    // Sequence is advanced only when the actual command image changes.
    // This keeps the command stable long enough for adapter ACK validation.
    L_Command_Changed :=
        (L_Command_Enable <> L_Last_Command_Enable[L_i]) OR
        (L_Setpoint_x10 <> L_Last_Command_Setpoint_x10[L_i]);

    IF L_Command_Changed THEN
        GVL_OPENTHERM_ADAPTER.G_Command[L_i].Sequence :=
            GVL_OPENTHERM_ADAPTER.G_Command[L_i].Sequence + 1;

        GVL_OPENTHERM_ADAPTER.G_Command[L_i].Last_Write_MS :=
            GVL_STATUS.G_System_Time_MS;

        L_Last_Command_Enable[L_i] := L_Command_Enable;
        L_Last_Command_Setpoint_x10[L_i] := L_Setpoint_x10;
    END_IF;

    // Command is valid only when the adapter confirms the current stable sequence.
    VO_OT_Command_Valid[L_i] :=
        L_Command_Enable AND
        GVL_OPENTHERM_ADAPTER.G_Status[L_i].Command_Ack AND
        (NOT GVL_OPENTHERM_ADAPTER.G_Status[L_i].Adapter_Error) AND
        GVL_OPENTHERM_ADAPTER.G_Status[L_i].Adapter_Online;

END_FOR;
          
END_FUNCTION_BLOCK

FUNCTION_BLOCK FB_Heating_Source_Stability_Observer
  VAR_INPUT
    VI_Enable : BOOL;
    VI_System_Time_MS : UDINT;
  END_VAR
  VAR
    L_i : INT;
    L_Last_Confidence : ARRAY[1..GVL_CONSTANTS.C_MAX_HEATING_CIRCUITS] OF REAL;
    L_Confidence_Delta : REAL;
    L_Confidence_Volatility : REAL;
    L_Source_Trust_Trend : REAL;
    L_Instability_Score : REAL;
  END_VAR

            // ==============================================================================
// Heating source stability observer
//
// Predictive observability-only layer.
//
// DOES NOT own runtime authority.
// DOES NOT own outputs.
// DOES NOT close valves.
// DOES NOT modify heating demand.
// DOES NOT override runtime decisions.
//
// Observes:
// - source switching frequency
// - fallback oscillation
// - degradation persistence
// - recovery trends
// - confidence volatility
//
// Publishes predictive instability semantics only.
//
// Reads only canonical runtime projection contracts.
// Does not depend on explainability publication topology.
// ==============================================================================



IF NOT VI_Enable THEN
    RETURN;
END_IF;

FOR L_i := 1 TO GVL_CONSTANTS.C_MAX_HEATING_CIRCUITS DO

    // ======================================================
    // VISIBILITY
    // ======================================================
    GVL_Heating_Source_Stability.G_State[L_i].Visible :=
        GVL_Heating_Runtime_Projection.G_Circuit_Projection[L_i].Visible;

    // ======================================================
    // EDGE COUNTING
    // ======================================================
    IF GVL_Heating_Runtime_Projection.G_Circuit_Projection[L_i].Source_Switched_Event THEN
        IF GVL_Heating_Source_Stability.G_State[L_i].Source_Switch_Count < 65535 THEN
            GVL_Heating_Source_Stability.G_State[L_i].Source_Switch_Count :=
                GVL_Heating_Source_Stability.G_State[L_i].Source_Switch_Count + 1;
        END_IF;

        GVL_Heating_Source_Stability.G_State[L_i].Last_Observation_MS :=
            VI_System_Time_MS;
    END_IF;

    IF GVL_Heating_Runtime_Projection.G_Circuit_Projection[L_i].Fallback_Activated_Event THEN
        IF GVL_Heating_Source_Stability.G_State[L_i].Fallback_Activation_Count < 65535 THEN
            GVL_Heating_Source_Stability.G_State[L_i].Fallback_Activation_Count :=
                GVL_Heating_Source_Stability.G_State[L_i].Fallback_Activation_Count + 1;
        END_IF;

        GVL_Heating_Source_Stability.G_State[L_i].Last_Observation_MS :=
            VI_System_Time_MS;
    END_IF;

    IF GVL_Heating_Runtime_Projection.G_Circuit_Projection[L_i].Fallback_Recovered_Event THEN
        IF GVL_Heating_Source_Stability.G_State[L_i].Fallback_Recovery_Count < 65535 THEN
            GVL_Heating_Source_Stability.G_State[L_i].Fallback_Recovery_Count :=
                GVL_Heating_Source_Stability.G_State[L_i].Fallback_Recovery_Count + 1;
        END_IF;

        GVL_Heating_Source_Stability.G_State[L_i].Last_Observation_MS :=
            VI_System_Time_MS;
    END_IF;

    IF GVL_Heating_Runtime_Projection.G_Circuit_Projection[L_i].Source_Loss_Event THEN
        IF GVL_Heating_Source_Stability.G_State[L_i].Source_Loss_Count < 65535 THEN
            GVL_Heating_Source_Stability.G_State[L_i].Source_Loss_Count :=
                GVL_Heating_Source_Stability.G_State[L_i].Source_Loss_Count + 1;
        END_IF;

        GVL_Heating_Source_Stability.G_State[L_i].Last_Observation_MS :=
            VI_System_Time_MS;
    END_IF;

    // ======================================================
    // CONFIDENCE VOLATILITY
    // ======================================================
    L_Confidence_Delta := ABS(
        GVL_Heating_Runtime_Projection.G_Circuit_Projection[L_i].Selected_Source_Confidence -
        L_Last_Confidence[L_i]
    );

    L_Confidence_Volatility :=
        GVL_Heating_Source_Stability.G_State[L_i].Confidence_Volatility * REAL#0.90 +
        L_Confidence_Delta * REAL#0.10;

    IF L_Confidence_Volatility < REAL#0.0 THEN
        L_Confidence_Volatility := REAL#0.0;
    ELSIF L_Confidence_Volatility > REAL#1.0 THEN
        L_Confidence_Volatility := REAL#1.0;
    END_IF;

    GVL_Heating_Source_Stability.G_State[L_i].Confidence_Volatility :=
        L_Confidence_Volatility;

    // ======================================================
    // SOURCE TRUST TREND
    // ======================================================
    L_Source_Trust_Trend :=
        GVL_Heating_Source_Stability.G_State[L_i].Source_Trust_Trend * REAL#0.95 +
        GVL_Heating_Runtime_Projection.G_Circuit_Projection[L_i].Selected_Source_Confidence * REAL#0.05;

    IF GVL_Heating_Runtime_Projection.G_Circuit_Projection[L_i].Source_Degraded THEN
        L_Source_Trust_Trend := L_Source_Trust_Trend * REAL#0.98;
    END_IF;

    IF L_Source_Trust_Trend < REAL#0.0 THEN
        L_Source_Trust_Trend := REAL#0.0;
    ELSIF L_Source_Trust_Trend > REAL#1.0 THEN
        L_Source_Trust_Trend := REAL#1.0;
    END_IF;

    GVL_Heating_Source_Stability.G_State[L_i].Source_Trust_Trend :=
        L_Source_Trust_Trend;

    // ======================================================
    // TREND OBSERVATION
    // ======================================================
    GVL_Heating_Source_Stability.G_State[L_i].Degraded_Trend_Visible :=
        GVL_Heating_Runtime_Projection.G_Circuit_Projection[L_i].Source_Degraded OR
        (GVL_Heating_Source_Stability.G_State[L_i].Fallback_Activation_Count >
         GVL_Heating_Source_Stability.G_State[L_i].Fallback_Recovery_Count);

    GVL_Heating_Source_Stability.G_State[L_i].Recovery_Trend_Visible :=
        (GVL_Heating_Source_Stability.G_State[L_i].Fallback_Recovery_Count > 0) AND
        (GVL_Heating_Source_Stability.G_State[L_i].Fallback_Recovery_Count >=
         GVL_Heating_Source_Stability.G_State[L_i].Fallback_Activation_Count);

    GVL_Heating_Source_Stability.G_State[L_i].Oscillation_Detected :=
        (GVL_Heating_Source_Stability.G_State[L_i].Source_Switch_Count >= 3) OR
        ((GVL_Heating_Source_Stability.G_State[L_i].Fallback_Activation_Count >= 2) AND
         (GVL_Heating_Source_Stability.G_State[L_i].Fallback_Recovery_Count >= 2));

    // ======================================================
    // INSTABILITY SCORE
    // ======================================================
    L_Instability_Score := REAL#0.0;

    IF GVL_Heating_Source_Stability.G_State[L_i].Oscillation_Detected THEN
        L_Instability_Score := L_Instability_Score + REAL#40.0;
    END_IF;

    IF GVL_Heating_Source_Stability.G_State[L_i].Degraded_Trend_Visible THEN
        L_Instability_Score := L_Instability_Score + REAL#30.0;
    END_IF;

    IF GVL_Heating_Source_Stability.G_State[L_i].Source_Loss_Count > 0 THEN
        L_Instability_Score := L_Instability_Score + REAL#30.0;
    END_IF;

    L_Instability_Score :=
        L_Instability_Score +
        (GVL_Heating_Source_Stability.G_State[L_i].Confidence_Volatility * REAL#20.0);

    IF L_Instability_Score > REAL#100.0 THEN
        L_Instability_Score := REAL#100.0;
    END_IF;

    GVL_Heating_Source_Stability.G_State[L_i].Instability_Score :=
        L_Instability_Score;

    GVL_Heating_Source_Stability.G_State[L_i].Instability_Attention :=
        L_Instability_Score >= REAL#60.0;

    // ======================================================
    // EXPLAINABILITY PUBLICATION
    // ======================================================
    IF GVL_Heating_Source_Stability.G_State[L_i].Source_Loss_Count > 0 THEN
        GVL_Heating_Source_Stability.G_State[L_i].Status_Code := 904;
        GVL_Heating_Source_Stability.G_State[L_i].Status_Text :=
            'Predictive source instability: source loss observed';

    ELSIF GVL_Heating_Source_Stability.G_State[L_i].Oscillation_Detected THEN
        GVL_Heating_Source_Stability.G_State[L_i].Status_Code := 903;
        GVL_Heating_Source_Stability.G_State[L_i].Status_Text :=
            'Predictive source instability: oscillation detected';

    ELSIF GVL_Heating_Source_Stability.G_State[L_i].Degraded_Trend_Visible THEN
        GVL_Heating_Source_Stability.G_State[L_i].Status_Code := 902;
        GVL_Heating_Source_Stability.G_State[L_i].Status_Text :=
            'Predictive source degradation trend observed';

    ELSE
        GVL_Heating_Source_Stability.G_State[L_i].Status_Code := 901;
        GVL_Heating_Source_Stability.G_State[L_i].Status_Text :=
            'Source stability nominal';
    END_IF;

    L_Last_Confidence[L_i] :=
        GVL_Heating_Runtime_Projection.G_Circuit_Projection[L_i].Selected_Source_Confidence;
END_FOR;

// >>> BULK_SYNC_ANCHOR: FB_Heating_Source_Stability_Observer <<<
          
END_FUNCTION_BLOCK

FUNCTION_BLOCK FB_Config_Simulation
  VAR_INPUT
    VI_Enable : BOOL;
    VI_Request : BOOL;
    VI_Confirm : BOOL;
  END_VAR
  VAR_OUTPUT
    VO_Executed : BOOL;
    VO_Result_OK : BOOL;
    VO_Error_Text : STRING(200);
  END_VAR
  VAR
    L_Error : BOOL;
  END_VAR

            // ==============================================================================
// Config simulation / validation function block
// Service/commissioning validation utility.
// Does NOT own runtime control and does NOT participate in heating phase runtime.
// ==============================================================================



VO_Executed := FALSE;
VO_Result_OK := GVL_CONFIG_SIMULATION.G_Simulation_Result_OK;
VO_Error_Text := GVL_CONFIG_SIMULATION.G_Simulation_Error_Text;

IF NOT VI_Enable THEN
    RETURN;
END_IF;

IF VI_Request AND VI_Confirm THEN

    L_Error := FALSE;
    VO_Result_OK := TRUE;
    VO_Error_Text := '';

    // Simulate INPUT constraints
    IF (GVL_CONFIG_CONTROL.STG_Reputation_Learning_Rate < 0.0) OR (GVL_CONFIG_CONTROL.STG_Reputation_Learning_Rate > 1.0) THEN
        VO_Result_OK := FALSE;
        VO_Error_Text := 'Invalid learning rate';
        L_Error := TRUE;
    END_IF;

    // Simulate SCENARIO logic
    IF GVL_CONFIG_CONTROL.STG_Night_Start_Hour = GVL_CONFIG_CONTROL.STG_Night_End_Hour THEN
        VO_Result_OK := FALSE;
        VO_Error_Text := 'Night window invalid';
        L_Error := TRUE;
    END_IF;

    // Simulate SAFETY
    IF GVL_CONFIG_CONTROL.STG_Stabilization_Delay_MS < 1000 THEN
        VO_Result_OK := FALSE;
        VO_Error_Text := 'Recovery delay too small';
        L_Error := TRUE;
    END_IF;

    // Simulate FAIL-SAFE policy
    IF NOT (
        GVL_CONFIG_CONTROL.STG_PLC_Inactive_Close_Gas OR
        GVL_CONFIG_CONTROL.STG_PLC_Inactive_Stop_Boiler OR
        GVL_CONFIG_CONTROL.STG_PLC_Inactive_Block_Heating OR
        GVL_CONFIG_CONTROL.STG_PLC_Inactive_Stop_Vent OR
        GVL_CONFIG_CONTROL.STG_PLC_Inactive_Block_Water
    ) THEN
        VO_Result_OK := FALSE;
        VO_Error_Text := 'Fail-safe disabled';
        L_Error := TRUE;
    END_IF;

    GVL_CONFIG_SIMULATION.G_Simulation_Result_OK := NOT L_Error;
    GVL_CONFIG_SIMULATION.G_Simulation_Error_Text := VO_Error_Text;
    GVL_CONFIG_SIMULATION.G_Simulation_Last_Run_MS := GVL_TIME_SERVICE.G_Now_MS;
    VO_Executed := TRUE;

END_IF;

// >>> BULK_SYNC_ANCHOR: FB_Config_Simulation <<<
          
END_FUNCTION_BLOCK

FUNCTION_BLOCK FB_DHW_Manager
  VAR_INPUT
    VI_System_Time_MS : UDINT;
    VI_Current_TOD : TOD;
    VI_IsActivePLC : BOOL;
    VI_Temp : REAL;
    VI_Pressure : REAL;
    VI_Config : ST_DHW_Config;
    VI_Current_Day_Of_Week : UINT;
    VI_Reset_Errors : BOOL;
    VI_Emergency_Stop : BOOL;
    VI_System_Mode : E_System_Operating_Mode;
    VI_IO_Modules_Online : ARRAY[1..GVL_CONSTANTS.C_MAX_MODULES] OF BOOL;
  END_VAR
  VAR_OUTPUT
    VO_Status : ST_DHW_Status;
    VO_Heating_Pump : BOOL;
    VO_Circ_Pump : BOOL;
  END_VAR
  VAR
    L_i : INT;
    L_Current_TOD : TOD;
    L_Legionella_Active : BOOL;
    L_Legionella_Timer : FB_System_Timer;
    L_Last_Good_Temp : REAL := 55.0;
    L_Legionella_Done_Today : BOOL;
    L_Last_Legionella_Day : UINT;
    fbTempValidator : FB_Analog_Validator;
    fbPressValidator : FB_Analog_Validator;
    L_Error_Latched : BOOL;
    L_Error_ID_Latched : WORD;
    L_Policy_Degraded : BOOL;
    L_Policy_Freeze_Protection : BOOL;
    L_Policy_Safe_Stop : BOOL;
    L_Target_Temp_Adjusted : REAL;
  END_VAR

            // >>> SYNC_TEST_MARKER_001 <<<


IF NOT VI_IsActivePLC THEN RETURN; END_IF;


GVL_STATE.G_DHW_IO_Fault := FALSE;
GVL_STATE.G_DHW_Sensor_Fault := FALSE;
GVL_STATE.G_DHW_Subsystem_Degraded := FALSE;

IF VI_Emergency_Stop THEN
    VO_Heating_Pump := FALSE;
    VO_Circ_Pump := FALSE;
    VO_Status.Warning := FALSE;
    VO_Status.Error := TRUE;
    VO_Status.Error_ID := TO_WORD(GVL_CONFIG.ERR_DHW_IO_OFFLINE); // временно используем общий аварийный код до детализации safety-кодов
    VO_Status.Heating_Pump_On := FALSE;
    VO_Status.Circ_Pump_On := FALSE;
    RETURN;
END_IF;

// Фиксация текущего времени
L_Current_TOD := VI_Current_TOD;

// ========================================
// DHW POLICY LAYER
// ========================================
L_Policy_Safe_Stop := (VI_System_Mode = E_System_Operating_Mode.MODE_SAFE_STOP);
L_Policy_Freeze_Protection := (VI_System_Mode = E_System_Operating_Mode.MODE_FREEZE_PROTECTION);
L_Policy_Degraded := (VI_System_Mode = E_System_Operating_Mode.MODE_DEGRADED);
L_Target_Temp_Adjusted := VI_Config.Target_Temp;
IF L_Policy_Degraded THEN
    L_Target_Temp_Adjusted := VI_Config.Target_Temp - VI_Config.Degraded_Target_Delta;
END_IF;

// ========================================
// DHW POLICY OVERRIDE
// ========================================
IF L_Policy_Safe_Stop THEN
    VO_Heating_Pump := FALSE;
    VO_Circ_Pump := FALSE;
    RETURN;
END_IF;

IF L_Policy_Freeze_Protection THEN
    VO_Heating_Pump := FALSE;
    VO_Circ_Pump := FALSE;
    RETURN;
END_IF;

// Сброс признака выполнения термодезинфекции при смене дня.
IF L_Last_Legionella_Day <> VI_Current_Day_Of_Week THEN
    L_Legionella_Done_Today := FALSE;
    L_Last_Legionella_Day := VI_Current_Day_Of_Week;
END_IF;

// Базовый сброс незащёлкнутых статусных флагов на текущий цикл.
// Критические ошибки ниже могут зафиксироваться и завершить выполнение через RETURN.
VO_Status.Warning := FALSE;
VO_Status.Error := FALSE;
VO_Status.Error_ID := 0;

// Сброс ошибок
IF VI_Reset_Errors THEN
    L_Error_Latched := FALSE;
    L_Error_ID_Latched := 0;
END_IF;

// Проверка связи с модулями ввода-вывода
FOR L_i := 1 TO GVL_CONSTANTS.C_MAX_MODULES DO
    IF NOT VI_IO_Modules_Online[L_i] THEN
        L_Error_Latched := TRUE;
        GVL_STATE.G_DHW_IO_Fault := TRUE;
        L_Error_ID_Latched := TO_WORD(GVL_CONFIG.ERR_DHW_IO_OFFLINE); // Потеря связи с модулями ввода-вывода
    END_IF;
END_FOR;

// 1. Обработка неисправностей датчиков и сервисных режимов (ТЗ 7.0)
fbTempValidator(
    VI_Value := VI_Temp,
    VI_Min_Valid := 0.0,
    VI_Max_Valid := 100.0,
    VI_Fallback_Mode := 0,
    VI_Default_Value := 55.0
);

fbPressValidator(
    VI_Value := VI_Pressure,
    VI_Min_Valid := 0.0,
    VI_Max_Valid := 10.0,
    VI_Fallback_Mode := 0
);

VO_Status.Temp := fbTempValidator.VO_Value;
VO_Status.Pressure := fbPressValidator.VO_Value;

// Сохраняем последнее достоверное значение температуры ГВС.
// Используется только для диагностики/сервиса, не для fallback-управления.
IF NOT fbTempValidator.VO_Error THEN
    L_Last_Good_Temp := VO_Status.Temp;
END_IF;

IF fbTempValidator.VO_Error THEN
    GVL_STATE.G_DHW_Sensor_Fault := TRUE;
    L_Error_Latched := TRUE;
    L_Error_ID_Latched := TO_WORD(GVL_CONFIG.ERR_DHW_TEMP_SENSOR_FAULT); // Критическая ошибка датчика температуры
ELSIF (VO_Status.Pressure < 1.0 OR VO_Status.Pressure > 4.0) AND NOT fbPressValidator.VO_Error THEN
    L_Error_Latched := TRUE;
    L_Error_ID_Latched := TO_WORD(GVL_CONFIG.ERR_DHW_PRESSURE_OUT_OF_RANGE); // Давление вне нормы
END_IF;

IF L_Error_Latched THEN
    // Критическая ошибка: переход в безопасное состояние с полной остановкой насосов.
    VO_Heating_Pump := FALSE;
    VO_Circ_Pump := FALSE;
    VO_Status.Warning := FALSE;
    VO_Status.Error := TRUE;
    VO_Status.Error_ID := L_Error_ID_Latched;
    VO_Status.Heating_Pump_On := FALSE;
    VO_Status.Circ_Pump_On := FALSE;
    RETURN;
END_IF;

// Ошибка датчика давления не останавливает ГВС,
// но переводит подсистему в режим предупреждения (degraded mode).
IF fbPressValidator.VO_Error THEN
    GVL_STATE.G_DHW_Sensor_Fault := TRUE;
    GVL_STATE.G_DHW_Subsystem_Degraded := TRUE;
    VO_Status.Warning := TRUE;
    VO_Status.Error := FALSE;
    VO_Status.Error_ID := TO_WORD(GVL_CONFIG.ERR_DHW_PRESSURE_SENSOR_FAULT);
END_IF;

// 2. Логика поддержания температуры воды в бойлере (Нагрев)
// На этом этапе FB уже выполняется только на активном ПЛК.
    
// Термическая дезинфекция (Легионелла)
IF VI_Config.Anti_Legionella_Enabled
   AND (VI_Current_Day_Of_Week = VI_Config.Anti_Legionella_Day)
   AND (L_Current_TOD >= TOD#02:00)
   AND (L_Current_TOD <= TOD#04:00)
   AND NOT L_Legionella_Done_Today THEN
    L_Legionella_Active := TRUE;
ELSE
    L_Legionella_Active := FALSE;
END_IF;

L_Legionella_Timer(IN := L_Legionella_Active AND VO_Status.Temp >= 70.0, PT := T#30m, VI_System_Time_MS := VI_System_Time_MS);
IF L_Legionella_Timer.Q THEN
    L_Legionella_Active := FALSE; // Дезинфекция завершена
    L_Legionella_Done_Today := TRUE; // Повторно в те же сутки не запускать
END_IF;

// Двухпозиционное регулирование с гистерезисом
IF L_Legionella_Active THEN
    IF VO_Status.Temp < 70.0 THEN
        VO_Heating_Pump := TRUE;
    ELSIF VO_Status.Temp > 72.0 THEN
        VO_Heating_Pump := FALSE;
    END_IF;
ELSE
    IF VO_Status.Temp < (L_Target_Temp_Adjusted - VI_Config.Hysteresis) THEN
        VO_Heating_Pump := TRUE;
    ELSIF VO_Status.Temp > (L_Target_Temp_Adjusted + VI_Config.Hysteresis) THEN
        VO_Heating_Pump := FALSE;
    END_IF;
END_IF;

// 3. Управление циркуляционным насосом ГВС по расписанию
// Рециркуляция обеспечивает мгновенное наличие горячей воды у потребителя
VO_Circ_Pump := SEL(VI_Config.Circulation_Schedule_Enabled AND NOT (VI_Config.Night_Mode_Enabled AND (L_Current_TOD < VI_Config.Circulation_Start OR L_Current_TOD > VI_Config.Circulation_End)), FALSE, TRUE);

// Формирование статусных данных для визуализации.
// К этому моменту статус уже консистентен:
// - Error = критическая ошибка с остановкой ГВС
// - Warning = деградация без остановки
VO_Status.Heating_Pump_On := VO_Heating_Pump;
VO_Status.Circ_Pump_On := VO_Circ_Pump;

// >>> BULK_SYNC_ANCHOR: FB_DHW_Manager <<<
          
END_FUNCTION_BLOCK

FUNCTION_BLOCK FB_CRC32_Calculator
  VAR_INPUT
    VI_Enable : BOOL := TRUE;
  END_VAR
  VAR_OUTPUT
    VO_CRC : DWORD;
  END_VAR
  VAR
    L_Table : ARRAY[0..255] OF DWORD;
    L_Initialized : BOOL := FALSE;
  END_VAR

            // Compatibility placeholder.
// Previous METHOD Calculate returned DWORD#0.
// Keep same behaviour without METHOD syntax for this CODESYS project format.
IF VI_Enable THEN
    VO_CRC := DWORD#0;
END_IF;
          
END_FUNCTION_BLOCK

FUNCTION_BLOCK FB_Heating_Runtime_Observability
  VAR_INPUT
    VI_Policy_Active : BOOL;
    VI_Freeze_Bypass_Active : BOOL;
    VI_DHW_Bypass_Active : BOOL;
    VI_Budget_Max : REAL;
    VI_Budget_Used : REAL;
    VI_Requested : ARRAY[1..GVL_CONSTANTS.C_MAX_MANIFOLDS] OF BOOL;
    VI_Allowed : ARRAY[1..GVL_CONSTANTS.C_MAX_MANIFOLDS] OF BOOL;
    VI_Filtered : ARRAY[1..GVL_CONSTANTS.C_MAX_MANIFOLDS] OF BOOL;
    VI_Block_Reason : ARRAY[1..GVL_CONSTANTS.C_MAX_MANIFOLDS] OF E_Heating_Allocation_Block_Reason;
    VI_Effective_Priority : ARRAY[1..GVL_CONSTANTS.C_MAX_MANIFOLDS] OF INT;
    VI_Priority_Bridge_Active : BOOL;
    VI_Priority_Bias_Applied : ARRAY[1..GVL_CONSTANTS.C_MAX_MANIFOLDS] OF REAL;
    VI_Priority_Effective : ARRAY[1..GVL_CONSTANTS.C_MAX_MANIFOLDS] OF INT;
  END_VAR
  VAR
    L_i : INT;
    L_Policy_Target_Adjustment : REAL;
    L_Policy_Priority_Multiplier : REAL;
  END_VAR

            // ==============================================================================
// Heating runtime observability layer
//
// Projection/publication layer only.
//
// IMPORTANT:
// - does NOT own outputs;
// - does NOT control pumps/valves;
// - does NOT modify demand;
// - does NOT participate in runtime authority.
//
// Responsibility:
// - allocation snapshot publication;
// - policy diagnostics projection;
// - freeze/DHW bypass visibility;
// - runtime explainability;
// - bounded policy bridge visibility.
// ==============================================================================



GVL_STATE.G_Allocation_Policy_Active := VI_Policy_Active;
GVL_STATE.G_Allocation_Freeze_Bypass_Active := VI_Freeze_Bypass_Active;
GVL_STATE.G_Allocation_DHW_Bypass_Active := VI_DHW_Bypass_Active;

GVL_STATE.G_Allocation_Budget_Max := VI_Budget_Max;
GVL_STATE.G_Allocation_Budget_Used := VI_Budget_Used;

FOR L_i := 1 TO GVL_CONSTANTS.C_MAX_MANIFOLDS DO
    GVL_STATE.G_Allocation_Requested[L_i] := VI_Requested[L_i];
    GVL_STATE.G_Allocation_Allowed[L_i] := VI_Allowed[L_i];
    GVL_STATE.G_Allocation_Filtered[L_i] := VI_Filtered[L_i];

    GVL_STATE.G_Allocation_Block_Reason[L_i] := VI_Block_Reason[L_i];
    GVL_STATE.G_Allocation_Effective_Priority[L_i] := VI_Effective_Priority[L_i];

    GVL_STATE.G_Policy_Priority_Bias_Applied[L_i] := VI_Priority_Bias_Applied[L_i];
    GVL_STATE.G_Policy_Priority_Effective[L_i] := VI_Priority_Effective[L_i];
END_FOR;

GVL_STATE.G_Policy_Priority_Bridge_Active := VI_Priority_Bridge_Active;

// Bounded policy target bridge visibility.
// Mirrors the same clamp used by FB_Heating_System_Manager.
L_Policy_Target_Adjustment := GVL_HEATING_POLICY.G_Policy_Target_Adjustment;
IF L_Policy_Target_Adjustment > REAL#5.0 THEN
    L_Policy_Target_Adjustment := REAL#5.0;
ELSIF L_Policy_Target_Adjustment < REAL#-3.0 THEN
    L_Policy_Target_Adjustment := REAL#-3.0;
END_IF;

L_Policy_Priority_Multiplier := GVL_HEATING_POLICY.G_Policy_Priority_Multiplier;
IF L_Policy_Priority_Multiplier < REAL#0.3 THEN
    L_Policy_Priority_Multiplier := REAL#0.3;
ELSIF L_Policy_Priority_Multiplier > REAL#1.0 THEN
    L_Policy_Priority_Multiplier := REAL#1.0;
END_IF;

GVL_STATE.G_Policy_Target_Adjustment_Applied := L_Policy_Target_Adjustment;
GVL_STATE.G_Policy_Target_Adjustment_Active := ABS(L_Policy_Target_Adjustment) > REAL#0.001;
GVL_STATE.G_Policy_Priority_Multiplier_Applied := L_Policy_Priority_Multiplier;

// >>> BULK_SYNC_ANCHOR: FB_Heating_Runtime_Observability <<<
          
END_FUNCTION_BLOCK

FUNCTION_BLOCK FB_Heating_Circuit_Explainability_Adapter
  VAR_INPUT
    VI_Enable : BOOL;
  END_VAR
  VAR
    L_i : INT;
  END_VAR

            // ==============================================================================
// Heating circuit explainability adapter
//
// Projection-to-explainability adapter.
//
// DOES NOT own runtime authority.
// DOES NOT own outputs.
// DOES NOT close valves.
// DOES NOT modify heating demand.
// DOES NOT override runtime decisions.
//
// Reads canonical runtime projection contracts and publishes legacy-compatible
// circuit explainability surfaces for HMI/diagnostics/supervisory visibility.
// ==============================================================================



IF NOT VI_Enable THEN
    RETURN;
END_IF;

FOR L_i := 1 TO GVL_CONSTANTS.C_MAX_HEATING_CIRCUITS DO
    GVL_Heating_Circuit_Explainability.G_Source_Selection_Visible[L_i] :=
        GVL_Heating_Runtime_Projection.G_Circuit_Projection[L_i].Visible;

    GVL_Heating_Circuit_Explainability.G_Selected_Source_Code[L_i] :=
        GVL_Heating_Runtime_Projection.G_Circuit_Projection[L_i].Selected_Source_Code;

    CASE GVL_Heating_Runtime_Projection.G_Circuit_Projection[L_i].Selected_Source_Code OF
        1:
            GVL_Heating_Circuit_Explainability.G_Selected_Source_Text[L_i] := 'room';
        2:
            GVL_Heating_Circuit_Explainability.G_Selected_Source_Text[L_i] := 'floor';
    ELSE
        GVL_Heating_Circuit_Explainability.G_Selected_Source_Text[L_i] := 'none';
    END_CASE;

    GVL_Heating_Circuit_Explainability.G_Fallback_Active[L_i] :=
        GVL_Heating_Runtime_Projection.G_Circuit_Projection[L_i].Fallback_Active;

    GVL_Heating_Circuit_Explainability.G_Source_Degraded[L_i] :=
        GVL_Heating_Runtime_Projection.G_Circuit_Projection[L_i].Source_Degraded;

    GVL_Heating_Circuit_Explainability.G_Selected_Source_Confidence[L_i] :=
        GVL_Heating_Runtime_Projection.G_Circuit_Projection[L_i].Selected_Source_Confidence;

    // Primary/fallback confidence remain legacy-compatible fields. The runtime
    // projection intentionally exposes selected confidence only, so these fields
    // mirror the selected source confidence until a dedicated richer projection
    // contract is introduced.
    GVL_Heating_Circuit_Explainability.G_Primary_Source_Confidence[L_i] :=
        GVL_Heating_Runtime_Projection.G_Circuit_Projection[L_i].Selected_Source_Confidence;

    GVL_Heating_Circuit_Explainability.G_Fallback_Source_Confidence[L_i] :=
        GVL_Heating_Runtime_Projection.G_Circuit_Projection[L_i].Selected_Source_Confidence;

    GVL_Heating_Circuit_Explainability.G_Reason_Code[L_i] :=
        GVL_Heating_Runtime_Projection.G_Circuit_Projection[L_i].Reason_Code;

    GVL_Heating_Circuit_Explainability.G_Reason_Text[L_i] :=
        GVL_Heating_Runtime_Projection.G_Circuit_Projection[L_i].Reason_Text;

    GVL_Heating_Circuit_Explainability.G_Source_Switched_Event[L_i] :=
        GVL_Heating_Runtime_Projection.G_Circuit_Projection[L_i].Source_Switched_Event;

    GVL_Heating_Circuit_Explainability.G_Fallback_Activated_Event[L_i] :=
        GVL_Heating_Runtime_Projection.G_Circuit_Projection[L_i].Fallback_Activated_Event;

    GVL_Heating_Circuit_Explainability.G_Fallback_Recovered_Event[L_i] :=
        GVL_Heating_Runtime_Projection.G_Circuit_Projection[L_i].Fallback_Recovered_Event;

    GVL_Heating_Circuit_Explainability.G_Source_Loss_Event[L_i] :=
        GVL_Heating_Runtime_Projection.G_Circuit_Projection[L_i].Source_Loss_Event;

    GVL_Heating_Circuit_Explainability.G_Last_Event_MS[L_i] :=
        GVL_Heating_Runtime_Projection.G_Circuit_Projection[L_i].Last_Event_MS;

    GVL_Heating_Circuit_Explainability.G_Last_Event_Code[L_i] :=
        GVL_Heating_Runtime_Projection.G_Circuit_Projection[L_i].Last_Event_Code;

    GVL_Heating_Circuit_Explainability.G_Last_Event_Text[L_i] :=
        GVL_Heating_Runtime_Projection.G_Circuit_Projection[L_i].Last_Event_Text;
END_FOR;

// >>> BULK_SYNC_ANCHOR: FB_Heating_Circuit_Explainability_Adapter <<<
          
END_FUNCTION_BLOCK

FUNCTION_BLOCK FB_Sensor_Calibration_Processor
  VAR_INPUT
    VI_Raw_Value : REAL;
    VI_Record : ST_Sensor_Calibration_Record;
  END_VAR
  VAR_OUTPUT
    VO_Calibrated_Value : REAL;
  END_VAR

            VO_Calibrated_Value := (VI_Raw_Value * VI_Record.multiplier) + VI_Record.offset;
          
END_FUNCTION_BLOCK

FUNCTION_BLOCK FB_Diagnostics_RootCause
  VAR_INPUT
    VI_Emergency_Stop : BOOL;
    VI_Gas_Safety : BOOL;
    VI_IO_Failsafe : BOOL;
    VI_Cascade_Available : BOOL;
    VI_Cascade_Degraded : BOOL;
    VI_Cascade_Partial_Capacity : BOOL;
    VI_Cascade_No_Flame : BOOL;
    VI_Cascade_Transport_Degraded : BOOL;
    VI_Cascade_Ignition_Timeout : BOOL;
    VI_Cascade_Active_Boilers : UINT;
    VI_Cascade_Available_Boilers : UINT;
    VI_Boiler_OT_Online : ARRAY[1..GVL_CONSTANTS.C_MAX_BOILERS] OF BOOL;
    VI_Boiler_Error : ARRAY[1..GVL_CONSTANTS.C_MAX_BOILERS] OF BOOL;
    VI_Boiler_Flame : ARRAY[1..GVL_CONSTANTS.C_MAX_BOILERS] OF BOOL;
    VI_Boiler_OT_Command_Timeout : ARRAY[1..GVL_CONSTANTS.C_MAX_BOILERS] OF BOOL;
    VI_Boiler_OT_Heartbeat_Timeout : ARRAY[1..GVL_CONSTANTS.C_MAX_BOILERS] OF BOOL;
    VI_Boiler_OT_Adapter_Error : ARRAY[1..GVL_CONSTANTS.C_MAX_BOILERS] OF BOOL;
    VI_Manifold_Pumps : ARRAY[1..GVL_CONSTANTS.C_MAX_MANIFOLDS] OF BOOL;
    VI_Manifold_Valves : ARRAY[1..GVL_CONSTANTS.C_MAX_MANIFOLDS] OF REAL;
    VI_Sensor_Error : BOOL;
    VI_Supply_Temps : ARRAY[1..GVL_CONSTANTS.C_MAX_MANIFOLDS] OF REAL;
    VI_Target_Supply : REAL;
    VI_Demand_Map : ARRAY[1..GVL_CONSTANTS.C_MAX_MANIFOLDS] OF BOOL;
  END_VAR
  VAR_OUTPUT
    VO_RootCause : E_Heating_RootCause;
    VO_Confidence : REAL;
    VO_Error_Score : REAL;
    VO_Reason_Code : INT;
    VO_Reason_Text : STRING(128);
  END_VAR
  VAR
    L_i : INT;
    L_AnyBoilerOnline : BOOL;
    L_AnyBoilerError : BOOL;
    L_AnyFlame : BOOL;
    L_AnyCommandTimeout : BOOL;
    L_AnyHeartbeatTimeout : BOOL;
    L_AnyAdapterError : BOOL;
    L_AnyDemand : BOOL;
    L_AnyPumpOn : BOOL;
    L_AnyValveOpen : BOOL;
    L_LowSupply : BOOL;
    L_CascadeSemanticKnown : BOOL;
  END_VAR

            // ==============================================================================
// Heating root-cause inference engine
// Internal diagnostics core.
// Does NOT own explainability publication or runtime control.
// ==============================================================================



// ======================================================
// DEFAULTS
// ======================================================
VO_RootCause := E_Heating_RootCause.RC_NONE;
VO_Confidence := 1.0;
VO_Error_Score := 0.0;
VO_Reason_Code := 0;
VO_Reason_Text := 'Heating inference OK';

// ======================================================
// SAFETY / GLOBAL BLOCKS
// ======================================================
IF VI_Emergency_Stop THEN
    VO_RootCause := E_Heating_RootCause.RC_EMERGENCY_STOP;
    VO_Confidence := 1.0;
    VO_Error_Score := 1.0;
    VO_Reason_Code := 10;
    VO_Reason_Text := 'Emergency stop active';
    RETURN;
END_IF;

IF VI_Gas_Safety THEN
    VO_RootCause := E_Heating_RootCause.RC_GAS_SAFETY;
    VO_Confidence := 1.0;
    VO_Error_Score := 1.0;
    VO_Reason_Code := 20;
    VO_Reason_Text := 'Gas safety active';
    RETURN;
END_IF;

IF VI_IO_Failsafe THEN
    VO_RootCause := E_Heating_RootCause.RC_IO_OFFLINE;
    VO_Confidence := 1.0;
    VO_Error_Score := 1.0;
    VO_Reason_Code := 30;
    VO_Reason_Text := 'Heating IO failsafe active';
    RETURN;
END_IF;

// ======================================================
// AGGREGATE LEGACY / LOW-LEVEL FLAGS
// ======================================================
L_AnyBoilerOnline := FALSE;
L_AnyBoilerError := FALSE;
L_AnyFlame := FALSE;
L_AnyCommandTimeout := FALSE;
L_AnyHeartbeatTimeout := FALSE;
L_AnyAdapterError := FALSE;

FOR L_i := 1 TO GVL_CONSTANTS.C_MAX_BOILERS DO
    IF VI_Boiler_OT_Online[L_i] THEN
        L_AnyBoilerOnline := TRUE;
    END_IF;

    IF VI_Boiler_Error[L_i] THEN
        L_AnyBoilerError := TRUE;
    END_IF;

    IF VI_Boiler_Flame[L_i] THEN
        L_AnyFlame := TRUE;
    END_IF;

    IF VI_Boiler_OT_Command_Timeout[L_i] THEN
        L_AnyCommandTimeout := TRUE;
    END_IF;

    IF VI_Boiler_OT_Heartbeat_Timeout[L_i] THEN
        L_AnyHeartbeatTimeout := TRUE;
    END_IF;

    IF VI_Boiler_OT_Adapter_Error[L_i] THEN
        L_AnyAdapterError := TRUE;
    END_IF;
END_FOR;

L_AnyDemand := FALSE;
L_AnyPumpOn := FALSE;
L_AnyValveOpen := FALSE;
L_LowSupply := FALSE;

FOR L_i := 1 TO GVL_CONSTANTS.C_MAX_MANIFOLDS DO
    IF VI_Demand_Map[L_i] THEN
        L_AnyDemand := TRUE;
    END_IF;

    IF VI_Manifold_Pumps[L_i] THEN
        L_AnyPumpOn := TRUE;
    END_IF;

    IF VI_Manifold_Valves[L_i] > 5.0 THEN
        L_AnyValveOpen := TRUE;
    END_IF;

    IF VI_Demand_Map[L_i] AND (VI_Supply_Temps[L_i] < (VI_Target_Supply - 2.0)) THEN
        L_LowSupply := TRUE;
    END_IF;
END_FOR;

L_CascadeSemanticKnown :=
    VI_Cascade_Available OR
    VI_Cascade_Degraded OR
    VI_Cascade_Partial_Capacity OR
    VI_Cascade_No_Flame OR
    VI_Cascade_Transport_Degraded OR
    VI_Cascade_Ignition_Timeout OR
    (VI_Cascade_Active_Boilers > 0) OR
    (VI_Cascade_Available_Boilers > 0);

// ======================================================
// MODERN CASCADE / OPENTHERM SEMANTICS
// ======================================================
IF L_CascadeSemanticKnown THEN

    IF NOT VI_Cascade_Available THEN
        VO_RootCause := E_Heating_RootCause.RC_BOILER_OFFLINE;
        VO_Confidence := 0.95;
        VO_Error_Score := 0.95;
        VO_Reason_Code := 100;
        VO_Reason_Text := 'Heating cascade unavailable';
        RETURN;
    END_IF;

    IF VI_Cascade_Transport_Degraded THEN
        IF L_AnyHeartbeatTimeout THEN
            VO_RootCause := E_Heating_RootCause.RC_IO_OFFLINE;
            VO_Confidence := 0.90;
            VO_Error_Score := 0.90;
            VO_Reason_Code := 210;
            VO_Reason_Text := 'OpenTherm heartbeat timeout';
            RETURN;
        END_IF;

        IF L_AnyCommandTimeout THEN
            VO_RootCause := E_Heating_RootCause.RC_IO_OFFLINE;
            VO_Confidence := 0.85;
            VO_Error_Score := 0.85;
            VO_Reason_Code := 220;
            VO_Reason_Text := 'OpenTherm command ACK timeout';
            RETURN;
        END_IF;

        IF L_AnyAdapterError THEN
            VO_RootCause := E_Heating_RootCause.RC_IO_OFFLINE;
            VO_Confidence := 0.85;
            VO_Error_Score := 0.85;
            VO_Reason_Code := 230;
            VO_Reason_Text := 'OpenTherm adapter error';
            RETURN;
        END_IF;

        VO_RootCause := E_Heating_RootCause.RC_IO_OFFLINE;
        VO_Confidence := 0.75;
        VO_Error_Score := 0.75;
        VO_Reason_Code := 200;
        VO_Reason_Text := 'OpenTherm transport degraded';
        RETURN;
    END_IF;

    IF VI_Cascade_Ignition_Timeout THEN
        VO_RootCause := E_Heating_RootCause.RC_NO_FLAME;
        VO_Confidence := 0.90;
        VO_Error_Score := 0.90;
        VO_Reason_Code := 300;
        VO_Reason_Text := 'Boiler ignition timeout';
        RETURN;
    END_IF;

    IF VI_Cascade_No_Flame THEN
        VO_RootCause := E_Heating_RootCause.RC_NO_FLAME;
        VO_Confidence := 0.80;
        VO_Error_Score := 0.80;
        VO_Reason_Code := 310;
        VO_Reason_Text := 'Cascade active but no flame';
        RETURN;
    END_IF;

    IF VI_Cascade_Partial_Capacity THEN
        VO_RootCause := E_Heating_RootCause.RC_LOW_SUPPLY_TEMP;
        VO_Confidence := 0.60;
        VO_Error_Score := 0.40;
        VO_Reason_Code := 500;
        VO_Reason_Text := 'Partial cascade capacity';
        RETURN;
    END_IF;
END_IF;

// ======================================================
// LEGACY BOILER / TRANSPORT FALLBACK
// ======================================================
IF NOT L_AnyBoilerOnline THEN
    VO_RootCause := E_Heating_RootCause.RC_BOILER_OFFLINE;
    VO_Confidence := 0.90;
    VO_Error_Score := 0.90;
    VO_Reason_Code := 110;
    VO_Reason_Text := 'No boiler online';
    RETURN;
END_IF;

IF L_AnyBoilerError THEN
    VO_RootCause := E_Heating_RootCause.RC_BOILER_ERROR;
    VO_Confidence := 0.90;
    VO_Error_Score := 0.90;
    VO_Reason_Code := 120;
    VO_Reason_Text := 'Boiler error active';
    RETURN;
END_IF;

IF L_AnyDemand AND NOT L_AnyFlame THEN
    VO_RootCause := E_Heating_RootCause.RC_NO_FLAME;
    VO_Confidence := 0.80;
    VO_Error_Score := 0.80;
    VO_Reason_Code := 130;
    VO_Reason_Text := 'Demand active but no flame';
    RETURN;
END_IF;

// ======================================================
// HYDRAULICS
// ======================================================
IF L_AnyDemand THEN
    IF NOT L_AnyPumpOn THEN
        VO_RootCause := E_Heating_RootCause.RC_PUMP_FAILURE;
        VO_Confidence := 0.80;
        VO_Error_Score := 0.80;
        VO_Reason_Code := 400;
        VO_Reason_Text := 'Demand active but manifold pumps are off';
        RETURN;
    END_IF;

    IF NOT L_AnyValveOpen THEN
        VO_RootCause := E_Heating_RootCause.RC_VALVES_CLOSED;
        VO_Confidence := 0.80;
        VO_Error_Score := 0.80;
        VO_Reason_Code := 410;
        VO_Reason_Text := 'Demand active but manifold valves are closed';
        RETURN;
    END_IF;
END_IF;

// ======================================================
// THERMAL TRANSFER
// ======================================================
IF L_AnyDemand AND L_LowSupply THEN
    VO_RootCause := E_Heating_RootCause.RC_NO_HEAT_TRANSFER;
    VO_Confidence := 0.70;
    VO_Error_Score := 0.70;
    VO_Reason_Code := 420;
    VO_Reason_Text := 'Supply temperature below target under demand';
    RETURN;
END_IF;

// ======================================================
// SENSORS
// ======================================================
IF VI_Sensor_Error THEN
    VO_RootCause := E_Heating_RootCause.RC_SENSOR_ERROR;
    VO_Confidence := 0.70;
    VO_Error_Score := 0.70;
    VO_Reason_Code := 450;
    VO_Reason_Text := 'Heating sensor error active';
    RETURN;
END_IF;

// ======================================================
// NORMAL
// ======================================================
VO_RootCause := E_Heating_RootCause.RC_NONE;
VO_Confidence := 1.0;
VO_Error_Score := 0.0;
VO_Reason_Code := 0;
VO_Reason_Text := 'Heating inference OK';
          
END_FUNCTION_BLOCK

FUNCTION_BLOCK FB_Water_Leakage_Manager
  VAR_INPUT
    VI_System_Time_MS : UDINT;
    VI_IsActivePLC : BOOL;
    VI_Config : ST_Flood_Global_Config;
  END_VAR
  VAR_OUTPUT
    VO_Status_Msg : STRING(200);
    VO_Leak_Detected : BOOL;
    VO_Leak_Warning_Level : BOOL;
  END_VAR
  VAR_IN_OUT
    VI_Sensors : ARRAY[1..GVL_CONSTANTS.C_MAX_FLOOD_SENSORS] OF BOOL;
  END_VAR
  VAR
    L_i : INT;
    L_Sensor_Timers : ARRAY[1..GVL_CONSTANTS.C_MAX_FLOOD_SENSORS] OF FB_System_Timer;
    L_Any_Leak : BOOL;
    L_Any_Warning : BOOL;
  END_VAR

            IF NOT VI_IsActivePLC THEN RETURN; END_IF;

L_Any_Leak := FALSE;
L_Any_Warning := FALSE;

FOR L_i := 1 TO GVL_CONSTANTS.C_MAX_FLOOD_SENSORS DO
    L_Sensor_Timers[L_i](
        IN := VI_Sensors[L_i],
        PT := TO_TIME(VI_Config.min_duration_ms + VI_Config.warning_duration_ms),
        VI_System_Time_MS := VI_System_Time_MS
    );

    IF L_Sensor_Timers[L_i].ET >= TO_TIME(VI_Config.min_duration_ms) THEN
        L_Any_Warning := TRUE;

        IF L_Sensor_Timers[L_i].Q THEN
            L_Any_Leak := TRUE;
        END_IF;
    END_IF;
END_FOR;

// Manual latch instead of RS
IF GVL_INTENT_USER.I_Reset_Errors THEN
    VO_Leak_Detected := FALSE;
ELSIF L_Any_Leak THEN
    VO_Leak_Detected := TRUE;
END_IF;

VO_Leak_Warning_Level := L_Any_Warning;

IF VO_Leak_Detected THEN
    VO_Status_Msg := 'АВАРИЯ: ПРОТЕЧКА ВОДЫ.';
ELSIF L_Any_Warning THEN
    VO_Status_Msg := 'ПРЕДУПРЕЖДЕНИЕ: ОБНАРУЖЕНА ВОДА.';
ELSE
    VO_Status_Msg := 'Система контроля протечек в норме';
END_IF;
// >>> BULK_SYNC_ANCHOR: FB_Water_Leakage_Manager <<<
          
END_FUNCTION_BLOCK

FUNCTION_BLOCK FB_Heating_Runtime_Explainability_Publisher
  VAR_INPUT
    VI_Enable : BOOL;
    VI_System_Time_MS : UDINT;
    VI_Runtime_Context : ST_Heating_Runtime_Context;
    VI_Runtime_Observation_Valid : BOOL;
    VI_Runtime_Observer_Fault : BOOL;
    VI_Runtime_Status_Code : UINT;
    VI_Runtime_Status_Text : STRING(128);
  END_VAR
  VAR_OUTPUT
    VO_Phase_Event : ST_Heating_Runtime_Phase_Event;
    VO_Anomaly : ST_Heating_Runtime_Anomaly;
    VO_Blackbox_Event : ST_Heating_Runtime_Blackbox_Event;
    VO_Blackbox_Timeline : ST_Heating_Runtime_Blackbox_Timeline;
    VO_Event_Buffer : ST_Heating_Runtime_Event_Buffer;
    VO_Adaptive_Intelligence : ST_Heating_Runtime_Adaptive_Intelligence;
    VO_Causality_Graph : ST_Heating_Runtime_Causality_Graph;
    VO_Integration_Bridge : ST_Heating_Runtime_Integration_Bridge;
    VO_Predictive_State : ST_Heating_Runtime_Predictive_State;
    VO_Execution_Timeline : ST_Heating_Runtime_Execution_Timeline;
    VO_Phase_Transition : ST_Heating_Runtime_Phase_Transition;
    VO_Publication_Valid : BOOL;
  END_VAR
  VAR
    L_Sequencing_Valid : BOOL;
    L_Ownership_Valid : BOOL;
    L_Synchronization_Valid : BOOL;
    L_Runtime_Degraded : BOOL;
    L_Status_Code : UINT;
  END_VAR

            L_Sequencing_Valid := VI_Runtime_Context.DHW_Before_Heating_Valid AND VI_Runtime_Context.State_Publication_Before_Diagnostics_Valid;
L_Ownership_Valid := VI_Runtime_Context.OpenTherm_Ownership_Valid AND VI_Runtime_Context.Cascade_Ownership_Valid AND VI_Runtime_Context.Safety_Isolation_Valid;
L_Synchronization_Valid := VI_Runtime_Context.Output_Projection_Last_Valid;
L_Runtime_Degraded := VI_Runtime_Observer_Fault OR NOT VI_Runtime_Observation_Valid;
L_Status_Code := VI_Runtime_Status_Code;

// Phase event
VO_Phase_Event.Phase := VI_Runtime_Context.Current_Phase;
VO_Phase_Event.Event_Active := VI_Enable;
VO_Phase_Event.Event_Completed := VI_Runtime_Observation_Valid;
VO_Phase_Event.Event_Failed := VI_Runtime_Observer_Fault;
VO_Phase_Event.Start_Time_MS := VI_System_Time_MS;
VO_Phase_Event.End_Time_MS := VI_System_Time_MS;
VO_Phase_Event.Duration_MS := 0;
VO_Phase_Event.Ordering_Valid := VI_Runtime_Context.DHW_Before_Heating_Valid;
VO_Phase_Event.Isolation_Valid := VI_Runtime_Context.Diagnostics_Isolation_Valid;
VO_Phase_Event.Status_Code := L_Status_Code;
VO_Phase_Event.Status_Text := VI_Runtime_Status_Text;
VO_Phase_Event.Diagnostics_Visible := TRUE;
VO_Phase_Event.Explainability_Visible := TRUE;
VO_Phase_Event.Safety_Integrity_Valid := VI_Runtime_Context.Safety_Isolation_Valid;
VO_Phase_Event.OpenTherm_Ownership_Valid := VI_Runtime_Context.OpenTherm_Ownership_Valid;
VO_Phase_Event.Cascade_Ownership_Valid := VI_Runtime_Context.Cascade_Ownership_Valid;

// Phase transition snapshot
VO_Phase_Transition.Previous_Phase := VI_Runtime_Context.Current_Phase;
VO_Phase_Transition.Current_Phase := VI_Runtime_Context.Current_Phase;
VO_Phase_Transition.Next_Phase := VI_Runtime_Context.Current_Phase;
VO_Phase_Transition.Transition_Active := VI_Enable;
VO_Phase_Transition.Transition_Completed := VI_Runtime_Observation_Valid;
VO_Phase_Transition.Transition_Failed := VI_Runtime_Observer_Fault;
VO_Phase_Transition.Transition_Start_MS := VI_System_Time_MS;
VO_Phase_Transition.Transition_End_MS := VI_System_Time_MS;
VO_Phase_Transition.Transition_Duration_MS := 0;
VO_Phase_Transition.Sequencing_Valid := L_Sequencing_Valid;
VO_Phase_Transition.Ownership_Valid := L_Ownership_Valid;
VO_Phase_Transition.Synchronization_Valid := L_Synchronization_Valid;
VO_Phase_Transition.Status_Code := L_Status_Code;
VO_Phase_Transition.Status_Text := VI_Runtime_Status_Text;

// Anomaly
VO_Anomaly.Anomaly_Active := VI_Runtime_Observer_Fault;
VO_Anomaly.Anomaly_Acknowledged := FALSE;
VO_Anomaly.Anomaly_Cleared := NOT VI_Runtime_Observer_Fault;
VO_Anomaly.Runtime_Jitter_Detected := FALSE;
VO_Anomaly.Runtime_Latency_Detected := FALSE;
VO_Anomaly.Runtime_Degraded := L_Runtime_Degraded;
VO_Anomaly.Cascade_Degraded := NOT VI_Runtime_Context.Cascade_Ownership_Valid;
VO_Anomaly.Cascade_Boiler_Loss_Detected := FALSE;
VO_Anomaly.OpenTherm_Transport_Degraded := NOT VI_Runtime_Context.OpenTherm_Ownership_Valid;
VO_Anomaly.OpenTherm_Command_Invalid := FALSE;
VO_Anomaly.Diagnostics_Degraded := NOT VI_Runtime_Context.Diagnostics_Isolation_Valid;
VO_Anomaly.Explainability_Degraded := NOT VI_Runtime_Context.Explainability_Isolation_Valid;
VO_Anomaly.Sequencing_Invalid := NOT L_Sequencing_Valid;
VO_Anomaly.Ownership_Invalid := NOT L_Ownership_Valid;
VO_Anomaly.Synchronization_Invalid := NOT L_Synchronization_Valid;
VO_Anomaly.Severity_Level := SEL(VI_Runtime_Observer_Fault, 1, 900);
VO_Anomaly.Critical_Anomaly := VI_Runtime_Observer_Fault;
VO_Anomaly.Status_Code := L_Status_Code;
VO_Anomaly.Status_Text := VI_Runtime_Status_Text;

// Blackbox event
VO_Blackbox_Event.Event_ID := VI_System_Time_MS;
VO_Blackbox_Event.Event_Active := VI_Enable;
VO_Blackbox_Event.Runtime_Phase := VI_Runtime_Context.Current_Phase;
VO_Blackbox_Event.Event_Start_MS := VI_System_Time_MS;
VO_Blackbox_Event.Event_End_MS := VI_System_Time_MS;
VO_Blackbox_Event.Event_Duration_MS := 0;
VO_Blackbox_Event.Runtime_Degraded := L_Runtime_Degraded;
VO_Blackbox_Event.Runtime_Fault := VI_Runtime_Observer_Fault;
VO_Blackbox_Event.Cascade_Degraded := NOT VI_Runtime_Context.Cascade_Ownership_Valid;
VO_Blackbox_Event.Cascade_Boiler_Loss := FALSE;
VO_Blackbox_Event.OpenTherm_Degraded := NOT VI_Runtime_Context.OpenTherm_Ownership_Valid;
VO_Blackbox_Event.OpenTherm_Command_Invalid := FALSE;
VO_Blackbox_Event.Sequencing_Invalid := NOT L_Sequencing_Valid;
VO_Blackbox_Event.Ownership_Invalid := NOT L_Ownership_Valid;
VO_Blackbox_Event.Synchronization_Invalid := NOT L_Synchronization_Valid;
VO_Blackbox_Event.Root_Cause_Candidate := VI_Runtime_Observer_Fault;
VO_Blackbox_Event.Critical_Path := VI_Runtime_Observer_Fault;
VO_Blackbox_Event.Status_Code := L_Status_Code;
VO_Blackbox_Event.Status_Text := VI_Runtime_Status_Text;

// Blackbox timeline snapshot
VO_Blackbox_Timeline.Write_Index := 1;
VO_Blackbox_Timeline.Event_Count := 1;
VO_Blackbox_Timeline.Timeline_Overflow := FALSE;
VO_Blackbox_Timeline.Reconstruction_Visible := TRUE;
VO_Blackbox_Timeline.Forensic_Timeline_Visible := TRUE;
VO_Blackbox_Timeline.Root_Cause_Reconstructed := VI_Runtime_Observer_Fault;
VO_Blackbox_Timeline.Sequencing_Valid := L_Sequencing_Valid;
VO_Blackbox_Timeline.Ownership_Valid := L_Ownership_Valid;
VO_Blackbox_Timeline.Synchronization_Valid := L_Synchronization_Valid;
VO_Blackbox_Timeline.Events[1] := VO_Blackbox_Event;
VO_Blackbox_Timeline.Status_Code := L_Status_Code;
VO_Blackbox_Timeline.Status_Text := VI_Runtime_Status_Text;

// Runtime event buffer snapshot
VO_Event_Buffer.Write_Index := 1;
VO_Event_Buffer.Read_Index := 1;
VO_Event_Buffer.Event_Count := 1;
VO_Event_Buffer.Overflow := FALSE;
VO_Event_Buffer.Ordering_Integrity_Valid := L_Sequencing_Valid;
VO_Event_Buffer.Isolation_Integrity_Valid := VI_Runtime_Context.Diagnostics_Isolation_Valid;
VO_Event_Buffer.Lifecycle_Integrity_Valid := VI_Runtime_Observation_Valid;
VO_Event_Buffer.Diagnostics_Visibility_Valid := TRUE;
VO_Event_Buffer.Explainability_Visibility_Valid := TRUE;
VO_Event_Buffer.OpenTherm_Ownership_Valid := VI_Runtime_Context.OpenTherm_Ownership_Valid;
VO_Event_Buffer.Cascade_Ownership_Valid := VI_Runtime_Context.Cascade_Ownership_Valid;
VO_Event_Buffer.Safety_Ownership_Valid := VI_Runtime_Context.Safety_Isolation_Valid;
VO_Event_Buffer.Events[1] := VO_Phase_Event;
VO_Event_Buffer.Status_Code := L_Status_Code;
VO_Event_Buffer.Status_Text := VI_Runtime_Status_Text;

// Passive integration bridge
VO_Integration_Bridge.Shell_Ready := VI_Runtime_Observation_Valid;
VO_Integration_Bridge.Shell_Fault := VI_Runtime_Observer_Fault;
VO_Integration_Bridge.Shell_Contract_Valid := VI_Enable AND VI_Runtime_Observation_Valid;
VO_Integration_Bridge.Allow_DHW_Integration := VI_Runtime_Context.Allow_DHW_Phase;
VO_Integration_Bridge.Allow_Heating_Integration := VI_Runtime_Context.Allow_Heating_Phase;
VO_Integration_Bridge.Allow_Diagnostics_Integration := VI_Runtime_Context.Allow_Diagnostics_Phase;
VO_Integration_Bridge.Allow_Output_Projection_Integration := VI_Runtime_Context.Allow_Output_Projection_Phase;
VO_Integration_Bridge.Runtime_Ownership_Valid := TRUE;
VO_Integration_Bridge.Diagnostics_Ownership_Valid := VI_Runtime_Context.Diagnostics_Isolation_Valid;
VO_Integration_Bridge.Explainability_Ownership_Valid := VI_Runtime_Context.Explainability_Isolation_Valid;
VO_Integration_Bridge.OpenTherm_Ownership_Valid := VI_Runtime_Context.OpenTherm_Ownership_Valid;
VO_Integration_Bridge.Cascade_Ownership_Valid := VI_Runtime_Context.Cascade_Ownership_Valid;
VO_Integration_Bridge.Safety_Ownership_Valid := VI_Runtime_Context.Safety_Isolation_Valid;
VO_Integration_Bridge.DHW_Before_Heating_Valid := VI_Runtime_Context.DHW_Before_Heating_Valid;
VO_Integration_Bridge.Diagnostics_After_Publication_Valid := VI_Runtime_Context.State_Publication_Before_Diagnostics_Valid;
VO_Integration_Bridge.Output_Projection_Last_Valid := VI_Runtime_Context.Output_Projection_Last_Valid;
VO_Integration_Bridge.Governance_Locked := TRUE;
VO_Integration_Bridge.Runtime_Attachment_Allowed := FALSE;
VO_Integration_Bridge.Runtime_Attachment_Active := FALSE;
VO_Integration_Bridge.Integration_Status_Code := L_Status_Code;
VO_Integration_Bridge.Integration_Status_Text := VI_Runtime_Status_Text;
VO_Integration_Bridge.Diagnostics_Visible := TRUE;
VO_Integration_Bridge.Explainability_Visible := TRUE;
VO_Integration_Bridge.Current_Phase := VI_Runtime_Context.Current_Phase;
VO_Integration_Bridge.Runtime_Synchronized := L_Synchronization_Valid;

// Predictive state (passive only)
VO_Predictive_State.Predictive_Analytics_Visible := TRUE;
VO_Predictive_State.Predictive_Analytics_Degraded := L_Runtime_Degraded;
VO_Predictive_State.Predictive_Analytics_Attention := NOT VI_Runtime_Observation_Valid;
VO_Predictive_State.Runtime_Stable := NOT L_Runtime_Degraded;
VO_Predictive_State.Runtime_Stability_Score := SEL(L_Runtime_Degraded, 100, 900);
VO_Predictive_State.Runtime_Degradation_Observation := SEL(L_Runtime_Degraded, 0, 900);
VO_Predictive_State.Runtime_Failure_Observation := SEL(VI_Runtime_Observer_Fault, 0, 900);
VO_Predictive_State.Cascade_Degradation_Observation := SEL(VI_Runtime_Context.Cascade_Ownership_Valid, 900, 0);
VO_Predictive_State.Cascade_Degraded_Trend_Visible := TRUE;
VO_Predictive_State.OpenTherm_Instability_Observation := SEL(VI_Runtime_Context.OpenTherm_Ownership_Valid, 900, 0);
VO_Predictive_State.OpenTherm_Degraded_Trend_Visible := TRUE;
VO_Predictive_State.Sequencing_Observation := SEL(L_Sequencing_Valid, 900, 0);
VO_Predictive_State.Ownership_Observation := SEL(L_Ownership_Valid, 900, 0);
VO_Predictive_State.Synchronization_Observation := SEL(L_Synchronization_Valid, 900, 0);
VO_Predictive_State.Status_Code := L_Status_Code;
VO_Predictive_State.Status_Text := VI_Runtime_Status_Text;

// Execution timeline snapshot
VO_Execution_Timeline.Write_Index := 1;
VO_Execution_Timeline.Frame_Count := 1;
VO_Execution_Timeline.Timeline_Overflow := FALSE;
VO_Execution_Timeline.Sequencing_Valid := L_Sequencing_Valid;
VO_Execution_Timeline.Ownership_Valid := L_Ownership_Valid;
VO_Execution_Timeline.Synchronization_Valid := L_Synchronization_Valid;
VO_Execution_Timeline.Runtime_Jitter_Detected := FALSE;
VO_Execution_Timeline.Runtime_Latency_Detected := FALSE;
VO_Execution_Timeline.Runtime_Degraded := L_Runtime_Degraded;
VO_Execution_Timeline.Frames[1].Phase := VI_Runtime_Context.Current_Phase;
VO_Execution_Timeline.Frames[1].Frame_Started := VI_Enable;
VO_Execution_Timeline.Frames[1].Frame_Completed := VI_Runtime_Observation_Valid;
VO_Execution_Timeline.Frames[1].Frame_Failed := VI_Runtime_Observer_Fault;
VO_Execution_Timeline.Frames[1].Frame_Start_MS := VI_System_Time_MS;
VO_Execution_Timeline.Frames[1].Frame_End_MS := VI_System_Time_MS;
VO_Execution_Timeline.Frames[1].Frame_Duration_MS := 0;
VO_Execution_Timeline.Frames[1].Sequencing_Valid := L_Sequencing_Valid;
VO_Execution_Timeline.Frames[1].Ownership_Valid := L_Ownership_Valid;
VO_Execution_Timeline.Frames[1].Synchronization_Valid := L_Synchronization_Valid;
VO_Execution_Timeline.Frames[1].Runtime_Jitter_Detected := FALSE;
VO_Execution_Timeline.Frames[1].Runtime_Latency_Detected := FALSE;
VO_Execution_Timeline.Frames[1].Runtime_Degraded := L_Runtime_Degraded;
VO_Execution_Timeline.Frames[1].Status_Code := L_Status_Code;
VO_Execution_Timeline.Frames[1].Status_Text := VI_Runtime_Status_Text;
VO_Execution_Timeline.Status_Code := L_Status_Code;
VO_Execution_Timeline.Status_Text := VI_Runtime_Status_Text;

// Adaptive intelligence (passive only)
VO_Adaptive_Intelligence.Adaptive_Analytics_Visible := TRUE;
VO_Adaptive_Intelligence.Adaptive_Analytics_Degraded := L_Runtime_Degraded;
VO_Adaptive_Intelligence.Adaptive_Analytics_Attention := NOT VI_Runtime_Observation_Valid;
VO_Adaptive_Intelligence.Supervision_Confidence_Observation := SEL(L_Runtime_Degraded, 100, 900);
VO_Adaptive_Intelligence.Confidence_Degradation_Visible := L_Runtime_Degraded;
VO_Adaptive_Intelligence.Adaptive_Runtime_Observation := 1;
VO_Adaptive_Intelligence.Adaptive_Runtime_Stability_Observation := SEL(L_Runtime_Degraded, 100, 900);
VO_Adaptive_Intelligence.Runtime_Anomaly_Observation_Weight := 1;
VO_Adaptive_Intelligence.Cascade_Anomaly_Observation_Weight := 1;
VO_Adaptive_Intelligence.OpenTherm_Anomaly_Observation_Weight := 1;
VO_Adaptive_Intelligence.Diagnostics_Anomaly_Observation_Weight := 1;
VO_Adaptive_Intelligence.Predictive_Correlation_Observation := 1;
VO_Adaptive_Intelligence.Predictive_Correlation_Visible := TRUE;
VO_Adaptive_Intelligence.Sequencing_Confidence_Observation := SEL(L_Sequencing_Valid, 100, 900);
VO_Adaptive_Intelligence.Ownership_Confidence_Observation := SEL(L_Ownership_Valid, 100, 900);
VO_Adaptive_Intelligence.Synchronization_Confidence_Observation := SEL(L_Synchronization_Valid, 100, 900);
VO_Adaptive_Intelligence.Status_Code := L_Status_Code;
VO_Adaptive_Intelligence.Status_Text := VI_Runtime_Status_Text;

// Minimal causality graph snapshot
VO_Causality_Graph.Node_Count := 1;
VO_Causality_Graph.Edge_Count := 1;
VO_Causality_Graph.Graph_Active := TRUE;
VO_Causality_Graph.Graph_Degraded := L_Runtime_Degraded;
VO_Causality_Graph.Graph_Critical := VI_Runtime_Observer_Fault;
VO_Causality_Graph.Sequencing_Valid := L_Sequencing_Valid;
VO_Causality_Graph.Ownership_Valid := L_Ownership_Valid;
VO_Causality_Graph.Synchronization_Valid := L_Synchronization_Valid;
VO_Causality_Graph.Nodes[1].Node_ID := 1;
VO_Causality_Graph.Nodes[1].Node_Active := TRUE;
VO_Causality_Graph.Nodes[1].Runtime_Degraded := L_Runtime_Degraded;
VO_Causality_Graph.Nodes[1].Runtime_Fault := VI_Runtime_Observer_Fault;
VO_Causality_Graph.Nodes[1].Cascade_Degraded := NOT VI_Runtime_Context.Cascade_Ownership_Valid;
VO_Causality_Graph.Nodes[1].OpenTherm_Degraded := NOT VI_Runtime_Context.OpenTherm_Ownership_Valid;
VO_Causality_Graph.Nodes[1].Diagnostics_Degraded := NOT VI_Runtime_Context.Diagnostics_Isolation_Valid;
VO_Causality_Graph.Nodes[1].Explainability_Degraded := NOT VI_Runtime_Context.Explainability_Isolation_Valid;
VO_Causality_Graph.Nodes[1].Sequencing_Invalid := NOT L_Sequencing_Valid;
VO_Causality_Graph.Nodes[1].Ownership_Invalid := NOT L_Ownership_Valid;
VO_Causality_Graph.Nodes[1].Synchronization_Invalid := NOT L_Synchronization_Valid;
VO_Causality_Graph.Nodes[1].Severity_Level := SEL(VI_Runtime_Observer_Fault, 1, 900);
VO_Causality_Graph.Nodes[1].Root_Cause_Candidate := VI_Runtime_Observer_Fault;
VO_Causality_Graph.Nodes[1].Status_Code := L_Status_Code;
VO_Causality_Graph.Nodes[1].Status_Text := VI_Runtime_Status_Text;
VO_Causality_Graph.Edges[1].Source_Node_ID := 1;
VO_Causality_Graph.Edges[1].Target_Node_ID := 1;
VO_Causality_Graph.Edges[1].Edge_Active := TRUE;
VO_Causality_Graph.Edges[1].Propagation_Detected := L_Runtime_Degraded;
VO_Causality_Graph.Edges[1].Runtime_Propagation := L_Runtime_Degraded;
VO_Causality_Graph.Edges[1].Cascade_Propagation := NOT VI_Runtime_Context.Cascade_Ownership_Valid;
VO_Causality_Graph.Edges[1].OpenTherm_Propagation := NOT VI_Runtime_Context.OpenTherm_Ownership_Valid;
VO_Causality_Graph.Edges[1].Diagnostics_Propagation := NOT VI_Runtime_Context.Diagnostics_Isolation_Valid;
VO_Causality_Graph.Edges[1].Sequencing_Propagation := NOT L_Sequencing_Valid;
VO_Causality_Graph.Edges[1].Ownership_Propagation := NOT L_Ownership_Valid;
VO_Causality_Graph.Edges[1].Synchronization_Propagation := NOT L_Synchronization_Valid;
VO_Causality_Graph.Status_Code := L_Status_Code;
VO_Causality_Graph.Status_Text := VI_Runtime_Status_Text;

VO_Publication_Valid := VI_Enable;

// >>> BULK_SYNC_ANCHOR: FB_Heating_Runtime_Explainability_Publisher <<<
          
END_FUNCTION_BLOCK

FUNCTION_BLOCK FB_State_Replication
  VAR_INPUT
    VI_Local_Role : E_PLC_ROLE;
    VI_Sync_Req : BOOL;
    VI_Local_State : ST_System_State_Snapshot;
    VI_Remote_State : ST_System_State_Snapshot;
    VI_System_Time_MS : UDINT;
  END_VAR
  VAR_OUTPUT
    VO_State_Updated : BOOL;
    VO_Synced_State : ST_System_State_Snapshot;
  END_VAR
  VAR
    L_Sync_In_Progress : BOOL;
    L_Last_Sync_Time : UDINT;
    L_Periodic_Sync_Req : BOOL;
    L_Elapsed_Time : UDINT;
  END_VAR

            // Периодическая синхронизация (каждые 5 секунд)
L_Elapsed_Time := (SEL(VI_System_Time_MS >= L_Last_Sync_Time, VI_System_Time_MS - L_Last_Sync_Time, (4294967295 - L_Last_Sync_Time) + VI_System_Time_MS + 1));

IF L_Elapsed_Time > 5000 THEN
    L_Periodic_Sync_Req := TRUE;
    L_Last_Sync_Time := VI_System_Time_MS;
ELSE
    L_Periodic_Sync_Req := FALSE;
END_IF;

// State Replication Logic
// Синхронизация состояния между ПЛК (ТЗ 8.2)
IF (VI_Sync_Req OR L_Periodic_Sync_Req) AND NOT L_Sync_In_Progress THEN
    L_Sync_In_Progress := TRUE;
    
    // Разрешение конфликтов на основе версии состояния
    IF VI_Remote_State.Version > VI_Local_State.Version THEN
        VO_Synced_State := VI_Remote_State;
        VO_State_Updated := TRUE;
    ELSIF VI_Remote_State.Version = VI_Local_State.Version THEN
        // Если версии равны, приоритет у ведущего ПЛК
        IF VI_Local_Role = E_PLC_ROLE.ROLE_STANDBY THEN
            VO_Synced_State := VI_Remote_State;
            VO_State_Updated := TRUE;
        ELSE
            VO_Synced_State := VI_Local_State;
            VO_State_Updated := FALSE;
        END_IF;
    ELSE
        VO_Synced_State := VI_Local_State;
        VO_State_Updated := FALSE;
    END_IF;
ELSIF NOT (VI_Sync_Req OR L_Periodic_Sync_Req) THEN
    L_Sync_In_Progress := FALSE;
    VO_State_Updated := FALSE;
    VO_Synced_State := VI_Local_State;
END_IF;
          
END_FUNCTION_BLOCK

FUNCTION_BLOCK FB_Water_Output_Projection
  VAR_INPUT
    VI_Zone_Enable : ARRAY[1..32] OF BOOL;
    VI_Valve_35_Close : BOOL;
    VI_Valve_36_Close : BOOL;
  END_VAR
  VAR
    L_i : INT;
  END_VAR

            FOR L_i := 1 TO 32 DO
    GVL_WATER_OUTPUT.DO_Water_Zone_Enable[L_i] := VI_Zone_Enable[L_i];
END_FOR;

GVL_WATER_OUTPUT.DO_Water_Valve_35_Close := VI_Valve_35_Close;
GVL_WATER_OUTPUT.DO_Water_Valve_36_Close := VI_Valve_36_Close;

// >>> BULK_SYNC_ANCHOR: FB_Water_Output_Projection <<<
          
END_FUNCTION_BLOCK

FUNCTION_BLOCK FB_Distributed_Projection_Ownership_Runtime
  VAR_INPUT
    VI_Enable : BOOL;
    VI_System_Time_MS : UDINT;
  END_VAR
  VAR
    L_i : INT;
    L_Ownership : ST_Distributed_Projection_Ownership;
    L_Any_Conflict : BOOL;
    L_Any_Stale : BOOL;
    L_Any_Blocked : BOOL;
    L_Finalized_Runtime_Continuity : BOOL;
  END_VAR

            IF NOT VI_Enable THEN
    GVL_Distributed_Projection_Ownership.G_Runtime_Valid := FALSE;
    RETURN;
END_IF;

// Finalized runtime continuity proof chain.
L_Finalized_Runtime_Continuity :=
    GVL_SEMANTIC_PROGRESS.Semantic_Forward_Progress_Valid
    AND GVL_SEMANTIC_PROGRESS.Semantic_Execution_Continuity_OK
    AND NOT GVL_SEMANTIC_PROGRESS.Semantic_Progress_Lease_Expired
    AND NOT GVL_SEMANTIC_PROGRESS.Semantic_Progress_Quarantine_Active
    AND GVL_RUNTIME_SNAPSHOT.Snapshot_Frozen
    AND GVL_RUNTIME_SNAPSHOT.Snapshot_Publication_Allowed
    AND GVL_RUNTIME_SNAPSHOT.Snapshot_Copy_Valid
    AND GVL_RUNTIME_SNAPSHOT.Snapshot_Isolation_Valid
    AND NOT GVL_RUNTIME_SNAPSHOT.Snapshot_Mutation_Detected
    AND GVL_DISTRIBUTED_SNAPSHOT.Distributed_Publication_Reconciled
    AND GVL_DISTRIBUTED_SNAPSHOT.Distributed_Publication_Freeze_Valid
    AND GVL_DISTRIBUTED_SNAPSHOT.Distributed_Snapshot_Consistent
    AND GVL_DISTRIBUTED_COMMIT.Distributed_Commit_Valid
    AND GVL_DISTRIBUTED_COMMIT.Publication_Prepare_Valid
    AND GVL_DISTRIBUTED_COMMIT.Publication_Commit_Confirmed
    AND NOT GVL_DISTRIBUTED_COMMIT.Peer_Commit_Mismatch
    AND NOT GVL_DISTRIBUTED_COMMIT.Commit_Lease_Expired
    AND GVL_OUTPUT_EPOCH.Output_Publication_Valid
    AND GVL_OUTPUT_EPOCH.Output_Runtime_Epoch_Valid
    AND NOT GVL_OUTPUT_EPOCH.Output_Lease_Expired
    AND NOT GVL_OUTPUT_EPOCH.Output_Forced_Safe_Decay
    AND GVL_COMMAND_VERIFY.PreOutput_Barrier_OK
    AND NOT GVL_COMMAND_VERIFY.PreOutput_Block_IO;

FOR L_i := 1 TO 128 DO

    L_Ownership :=
        GVL_Distributed_Projection_Ownership.G_Projection_Ownership[L_i];

    IF L_Ownership.Ownership_Valid THEN

        L_Ownership.Runtime_System_Time_MS :=
            VI_System_Time_MS;

        // Ownership becomes stale if runtime sessions unhealthy.
        IF GVL_Runtime_Sessions.G_Any_Stale_Session THEN

            L_Ownership.Ownership_Stale := TRUE;
            L_Any_Stale := TRUE;

        END_IF;

        // Finalized continuity loss invalidates ownership.
        IF NOT L_Finalized_Runtime_Continuity THEN

            L_Ownership.Ownership_Stale := TRUE;
            L_Ownership.Projection_Blocked := TRUE;

            L_Any_Stale := TRUE;
            L_Any_Blocked := TRUE;

        END_IF;

        // Hard conflict prevention.
        IF GVL_Distributed_Runtime.G_Split_Brain_Suspected THEN

            L_Ownership.Ownership_Conflict := TRUE;
            L_Ownership.Projection_Blocked := TRUE;

            L_Any_Conflict := TRUE;
            L_Any_Blocked := TRUE;

        END_IF;

        // Distributed execution authority.
        IF GVL_Distributed_Authority.G_Authority_State.Authority_Master_Elected
           AND NOT L_Ownership.Ownership_Conflict
           AND NOT L_Ownership.Ownership_Stale
           AND L_Finalized_Runtime_Continuity THEN

            L_Ownership.Ownership_Granted := TRUE;
            L_Ownership.Distributed_Execution_Allowed := TRUE;
            L_Ownership.Distributed_Recovery_Allowed := TRUE;

            L_Ownership.Status_Code := 0;
            L_Ownership.Status_Text :=
                'Distributed projection ownership granted';

        ELSE

            L_Ownership.Ownership_Revoked := TRUE;
            L_Ownership.Projection_Blocked := TRUE;

            L_Any_Blocked := TRUE;

            L_Ownership.Status_Code := 2;
            L_Ownership.Status_Text :=
                'Distributed projection ownership blocked';

        END_IF;

        GVL_Distributed_Projection_Ownership.G_Projection_Ownership[L_i] :=
            L_Ownership;

    END_IF;

END_FOR;

GVL_Distributed_Projection_Ownership.G_Any_Ownership_Conflict :=
    L_Any_Conflict;

GVL_Distributed_Projection_Ownership.G_Any_Ownership_Stale :=
    L_Any_Stale;

GVL_Distributed_Projection_Ownership.G_Any_Projection_Blocked :=
    L_Any_Blocked;

GVL_Distributed_Projection_Ownership.G_Runtime_Valid := TRUE;
GVL_Distributed_Projection_Ownership.G_Last_Update_MS :=
    VI_System_Time_MS;

IF L_Any_Conflict THEN
    GVL_Distributed_Projection_Ownership.G_Status_Code := 3;
    GVL_Distributed_Projection_Ownership.G_Status_Text :=
        'Distributed projection ownership conflict detected';
ELSIF L_Any_Stale THEN
    GVL_Distributed_Projection_Ownership.G_Status_Code := 2;
    GVL_Distributed_Projection_Ownership.G_Status_Text :=
        'Distributed projection ownership stale';
ELSIF L_Any_Blocked THEN
    GVL_Distributed_Projection_Ownership.G_Status_Code := 1;
    GVL_Distributed_Projection_Ownership.G_Status_Text :=
        'Distributed projection ownership blocked';
ELSE
    GVL_Distributed_Projection_Ownership.G_Status_Code := 0;
    GVL_Distributed_Projection_Ownership.G_Status_Text :=
        'Distributed projection ownership healthy';
END_IF;
          
END_FUNCTION_BLOCK

FUNCTION_BLOCK FB_Heating_Runtime_Output_Projection_Phase
  VAR_INPUT
    VI_Enable : BOOL;
    VI_Zone_Valves : ARRAY[1..GVL_CONSTANTS.C_MAX_HEATING_CIRCUITS] OF BOOL;
    VI_Manifold_Pumps : ARRAY[1..GVL_CONSTANTS.C_MAX_MANIFOLDS] OF BOOL;
    VI_Manifold_Valves : ARRAY[1..GVL_CONSTANTS.C_MAX_MANIFOLDS] OF REAL;
    VI_DHW_Heating_Pump : BOOL;
    VI_DHW_Circ_Pump : BOOL;
    VI_Backup_Circulation_Pump : BOOL;
    VI_Electric_Heater_Enable : BOOL;
  END_VAR
  VAR_OUTPUT
    VO_Executed : BOOL;
    VO_Valid : BOOL;
  END_VAR
  VAR
    fbOutputProjection : FB_Heating_Output_Projection;
  END_VAR

            // ==============================================================================
// Heating runtime output projection phase
// Final phase wrapper around physical output projection.
// Does NOT calculate heating logic and does NOT publish state/status.
// ==============================================================================



VO_Executed := FALSE;
VO_Valid := FALSE;

IF NOT VI_Enable THEN
    RETURN;
END_IF;

fbOutputProjection(
    VI_Zone_Valves := VI_Zone_Valves,
    VI_Manifold_Pumps := VI_Manifold_Pumps,
    VI_Manifold_Valves := VI_Manifold_Valves,
    VI_DHW_Heating_Pump := VI_DHW_Heating_Pump,
    VI_DHW_Circ_Pump := VI_DHW_Circ_Pump,
    VI_Backup_Circulation_Pump := VI_Backup_Circulation_Pump,
    VI_Electric_Heater_Enable := VI_Electric_Heater_Enable
);

VO_Executed := TRUE;
VO_Valid := TRUE;

// >>> BULK_SYNC_ANCHOR: FB_Heating_Runtime_Output_Projection_Phase <<<
          
END_FUNCTION_BLOCK

FUNCTION_BLOCK FB_Gas_Smoke_Manager
  VAR_INPUT
    VI_System_Time_MS : UDINT;
    VI_IsActivePLC : BOOL;
    VI_Mute_Request : BOOL;
  END_VAR
  VAR_OUTPUT
    VO_Smoke_Detected : BOOL;
    VO_Gas_Detected : BOOL;
    VO_CO_Warning_Level : BOOL;
    VO_CO_Alarm_Level : BOOL;
    VO_Status_Msg : STRING(200);
  END_VAR
  VAR_IN_OUT
    VI_Methane_LEL : ARRAY[1..GVL_CONSTANTS.C_MAX_METHANE_SENSORS] OF REAL;
    VI_CO_PPM : ARRAY[1..GVL_CONSTANTS.C_MAX_CO_SENSORS] OF REAL;
    VI_Smoke_Sensors : ARRAY[1..GVL_CONSTANTS.C_MAX_SMOKE_SENSORS] OF BOOL;
  END_VAR
  VAR
    L_Methane_Max : REAL;
    L_CO_Max : REAL;
    L_Smoke_Count : UINT;
    L_Smoke_Active : BOOL;
    L_i : INT;
    L_CO_Timer_30ppm : FB_System_Timer;
    L_CO_Timer_70ppm : FB_System_Timer;
    L_CO_Timer_400ppm : FB_System_Timer;
    L_CO_Level_30 : BOOL;
    L_CO_Level_70 : BOOL;
    L_CO_Level_400 : BOOL;
    L_Smoke_Timer : ARRAY[1..GVL_CONSTANTS.C_MAX_SMOKE_SENSORS] OF FB_System_Timer;
  END_VAR

            IF NOT VI_IsActivePLC THEN RETURN; END_IF;

// Reset outputs
VO_Smoke_Detected := FALSE;
VO_Gas_Detected := FALSE;
VO_CO_Warning_Level := FALSE;
VO_CO_Alarm_Level := FALSE;
VO_Status_Msg := 'ОК';

// --- Methane ---
L_Methane_Max := 0.0;
FOR L_i := 1 TO GVL_CONSTANTS.C_MAX_METHANE_SENSORS DO
    IF VI_Methane_LEL[L_i] > L_Methane_Max THEN
        L_Methane_Max := VI_Methane_LEL[L_i];
    END_IF;
END_FOR;

IF L_Methane_Max >= 20.0 THEN
    VO_Gas_Detected := TRUE;
END_IF;

// --- CO ---
L_CO_Max := 0.0;
FOR L_i := 1 TO GVL_CONSTANTS.C_MAX_CO_SENSORS DO
    IF VI_CO_PPM[L_i] > L_CO_Max THEN
        L_CO_Max := VI_CO_PPM[L_i];
    END_IF;
END_FOR;

L_CO_Level_30 := (L_CO_Max >= 30.0);
L_CO_Level_70 := (L_CO_Max >= 70.0);
L_CO_Level_400 := (L_CO_Max >= 400.0);

L_CO_Timer_30ppm(IN := L_CO_Level_30, PT := T#8h, VI_System_Time_MS := VI_System_Time_MS);
L_CO_Timer_70ppm(IN := L_CO_Level_70, PT := T#1h, VI_System_Time_MS := VI_System_Time_MS);
L_CO_Timer_400ppm(IN := L_CO_Level_400, PT := T#15m, VI_System_Time_MS := VI_System_Time_MS);

IF L_CO_Timer_30ppm.Q THEN
    VO_CO_Warning_Level := TRUE;
END_IF;

IF L_CO_Timer_70ppm.Q OR L_CO_Timer_400ppm.Q THEN
    VO_CO_Alarm_Level := TRUE;
END_IF;

// --- Smoke ---
L_Smoke_Count := 0;
L_Smoke_Active := FALSE;

FOR L_i := 1 TO GVL_CONSTANTS.C_MAX_SMOKE_SENSORS DO
    L_Smoke_Timer[L_i](IN := VI_Smoke_Sensors[L_i], PT := T#30s, VI_System_Time_MS := VI_System_Time_MS);

    IF VI_Smoke_Sensors[L_i] THEN
        L_Smoke_Count := L_Smoke_Count + 1;
    END_IF;

    IF L_Smoke_Timer[L_i].Q OR (L_Smoke_Count >= 2) THEN
        L_Smoke_Active := TRUE;
    END_IF;
END_FOR;

IF L_Smoke_Active THEN
    VO_Smoke_Detected := TRUE;
END_IF;

// Status
IF VO_Smoke_Detected THEN
    VO_Status_Msg := 'ПОЖАР';
ELSIF VO_Gas_Detected THEN
    VO_Status_Msg := 'УТЕЧКА ГАЗА';
ELSIF VO_CO_Alarm_Level THEN
    VO_Status_Msg := 'КРИТИЧЕСКИЙ CO';
ELSIF VO_CO_Warning_Level THEN
    VO_Status_Msg := 'ПОВЫШЕННЫЙ CO';
ELSE
    VO_Status_Msg := 'ОК';
END_IF;
// >>> BULK_SYNC_ANCHOR: FB_Gas_Smoke_Manager <<<
          
END_FUNCTION_BLOCK

FUNCTION_BLOCK FB_Input_Quality_Observer
  VAR_INPUT
    VI_Enable : BOOL;
    VI_Value : REAL;
    VI_System_Time_MS : UDINT;
    VI_Spike_Threshold : REAL;
    VI_Stuck_Timeout_MS : UDINT;
  END_VAR
  VAR_OUTPUT
    VO_Quality : ST_Input_Quality_Record;
  END_VAR
  VAR
    L_Last_Value : REAL;
    L_Last_Change_MS : UDINT;
    L_Delta : REAL;
  END_VAR

            VO_Quality.Quality_Visible := VI_Enable;

IF NOT VI_Enable THEN
    RETURN;
END_IF;

VO_Quality.Value_Valid := TRUE;
VO_Quality.Value_Degraded := FALSE;
VO_Quality.Spike_Detected := FALSE;
VO_Quality.Stuck_Detected := FALSE;
VO_Quality.Confidence := REAL#1.0;
VO_Quality.Reason_Code := 0;
VO_Quality.Reason_Text := 'OK';

L_Delta := ABS(VI_Value - L_Last_Value);

IF L_Delta > VI_Spike_Threshold THEN
    VO_Quality.Spike_Detected := TRUE;
    VO_Quality.Value_Degraded := TRUE;
    VO_Quality.Confidence := REAL#0.4;
    VO_Quality.Reason_Code := 1;
    VO_Quality.Reason_Text := 'Spike detected';
END_IF;

IF L_Delta > REAL#0.05 THEN
    L_Last_Change_MS := VI_System_Time_MS;
END_IF;

IF (VI_System_Time_MS > L_Last_Change_MS) AND
   ((VI_System_Time_MS - L_Last_Change_MS) > VI_Stuck_Timeout_MS) THEN

    VO_Quality.Stuck_Detected := TRUE;
    VO_Quality.Value_Degraded := TRUE;

    IF VO_Quality.Confidence > REAL#0.6 THEN
        VO_Quality.Confidence := REAL#0.6;
    END_IF;

    IF VO_Quality.Reason_Code = 0 THEN
        VO_Quality.Reason_Code := 2;
        VO_Quality.Reason_Text := 'Sensor appears stuck';
    END_IF;
END_IF;

VO_Quality.Last_Value := VI_Value;
VO_Quality.Last_Change_MS := L_Last_Change_MS;

L_Last_Value := VI_Value;
          
END_FUNCTION_BLOCK

FUNCTION_BLOCK FB_Water_Valve_Feedback_Runtime
  VAR_INPUT
    VI_Enable : BOOL;
    VI_System_Time_MS : UDINT;
  END_VAR
  VAR
    L_i : INT;
    L_Output : ST_Water_Output_Projection_State;
    L_State : ST_Water_Valve_Feedback_State;
    L_Any_Degraded : BOOL;
    L_Any_Timeout : BOOL;
    L_Any_Conflict : BOOL;
  END_VAR

            IF NOT VI_Enable THEN
    GVL_Water_Valve_Feedback.G_Runtime_Valid := FALSE;
    RETURN;
END_IF;

FOR L_i := 1 TO GVL_CONSTANTS.C_MAX_FLOOD_SENSORS DO

    L_Output := GVL_Water_Output_Projection.G_Output_Projection_State[L_i];

    L_State := (Runtime_Valid := TRUE);

    L_State.Runtime_System_Time_MS := VI_System_Time_MS;
    L_State.Valve_Group_Id := L_Output.Valve_Group_Id;

    // Feedback integration hook.
    // Conservative observe-only mode until physical DI binding is connected.
    L_State.Feedback_Available := FALSE;

    // No forced degraded state in observe-only mode.
    IF L_State.Feedback_Available THEN

        IF L_State.Physical_Open_Feedback
           AND L_State.Physical_Closed_Feedback THEN

            L_State.Feedback_Conflict := TRUE;
            L_State.Valve_Degraded := TRUE;

        END_IF;

        L_State.Confirmed_Open :=
            L_State.Physical_Open_Feedback
            AND NOT L_State.Physical_Closed_Feedback;

        L_State.Confirmed_Closed :=
            L_State.Physical_Closed_Feedback
            AND NOT L_State.Physical_Open_Feedback;

    ELSE

        L_State.Confirmation_Unknown := TRUE;

    END_IF;

    IF L_State.Feedback_Conflict THEN
        L_State.Status_Code := 3;
        L_State.Status_Text :=
            'Valve feedback conflict detected';
    ELSIF L_State.Feedback_Timeout THEN
        L_State.Status_Code := 2;
        L_State.Status_Text :=
            'Valve feedback timeout';
    ELSIF L_State.Confirmation_Unknown THEN
        L_State.Status_Code := 1;
        L_State.Status_Text :=
            'Valve feedback unavailable';
    ELSE
        L_State.Status_Code := 0;
        L_State.Status_Text :=
            'Valve feedback healthy';
    END_IF;

    GVL_Water_Valve_Feedback.G_Valve_Feedback_State[L_i] :=
        L_State;

    L_Any_Degraded :=
        L_Any_Degraded
        OR L_State.Valve_Degraded;

    L_Any_Timeout :=
        L_Any_Timeout
        OR L_State.Feedback_Timeout;

    L_Any_Conflict :=
        L_Any_Conflict
        OR L_State.Feedback_Conflict;

END_FOR;

GVL_Water_Valve_Feedback.G_Any_Degraded :=
    L_Any_Degraded;

GVL_Water_Valve_Feedback.G_Any_Timeout :=
    L_Any_Timeout;

GVL_Water_Valve_Feedback.G_Any_Conflict :=
    L_Any_Conflict;

GVL_Water_Valve_Feedback.G_Runtime_Valid := TRUE;
GVL_Water_Valve_Feedback.G_Last_Update_MS := VI_System_Time_MS;

IF L_Any_Conflict THEN
    GVL_Water_Valve_Feedback.G_Status_Code := 3;
    GVL_Water_Valve_Feedback.G_Status_Text :=
        'Valve feedback conflicts detected';
ELSIF L_Any_Timeout THEN
    GVL_Water_Valve_Feedback.G_Status_Code := 2;
    GVL_Water_Valve_Feedback.G_Status_Text :=
        'Valve feedback degraded';
ELSIF L_Any_Degraded THEN
    GVL_Water_Valve_Feedback.G_Status_Code := 1;
    GVL_Water_Valve_Feedback.G_Status_Text :=
        'Valve diagnostics degraded';
ELSE
    GVL_Water_Valve_Feedback.G_Status_Code := 0;
    GVL_Water_Valve_Feedback.G_Status_Text :=
        'Valve feedback runtime healthy';
END_IF;
          
END_FUNCTION_BLOCK

FUNCTION_BLOCK FB_Water_Output_Projector
  VAR_INPUT
    VI_Enable : BOOL;
    VI_System_Time_MS : UDINT;
  END_VAR
  VAR
    L_i : INT;
    L_Authority : ST_Water_Isolation_Authority_State;
    L_Valve : ST_Water_Valve_Runtime_State;
    L_Output : ST_Water_Output_Projection_State;
    L_Any_Projected : BOOL;
    L_Any_Denied : BOOL;
    L_Global_Fallback : BOOL;
  END_VAR

            IF NOT VI_Enable THEN
    GVL_Water_Output_Projection.G_Runtime_Valid := FALSE;
    RETURN;
END_IF;

L_Any_Projected := FALSE;
L_Any_Denied := FALSE;
L_Global_Fallback := FALSE;

FOR L_i := 1 TO GVL_CONSTANTS.C_MAX_FLOOD_SENSORS DO

    L_Authority := GVL_Water_Isolation_Authority.G_Authority_State[L_i];
    L_Valve := GVL_Water_Valve_Runtime.G_Valve_Runtime_State[L_i];

    L_Output.Projection_Valid := FALSE;
    L_Output.Projection_Valid := TRUE;
    L_Output.Projection_System_Time_MS := VI_System_Time_MS;
    L_Output.Output_Owner_Valid := TRUE;
    L_Output.Output_Owner_Id := TO_UINT(L_i);
    L_Output.Valve_Id := L_Valve.Valve_Id;
    L_Output.Valve_Group_Id := L_Valve.Valve_Group_Id;
    L_Output.Selective_Authority_Allowed := L_Authority.Selective_Authority_Allowed;
    L_Output.Global_Fallback_Required := L_Authority.Global_Fallback_Required;
    L_Output.Authority_Valid := L_Authority.Decision_Valid;

    IF L_Output.Global_Fallback_Required THEN
        L_Output.Projection_Allowed := TRUE;
        L_Output.Physical_Close_Project := TRUE;
        L_Output.Expected_Closed := TRUE;
        L_Output.Projection_Code := 1;
        L_Output.Projection_Text := 'Global fallback output projection active';
        L_Global_Fallback := TRUE;
    ELSIF L_Output.Selective_Authority_Allowed AND L_Output.Authority_Valid THEN
        L_Output.Projection_Allowed := TRUE;
        L_Output.Physical_Close_Project := TRUE;
        L_Output.Expected_Closed := TRUE;
        L_Output.Projection_Code := 10;
        L_Output.Projection_Text := 'Selective authority output projection active';
    ELSE
        L_Output.Projection_Denied := TRUE;
        L_Output.Projection_Code := 100;
        L_Output.Projection_Text := 'Projection denied';
        L_Any_Denied := TRUE;
    END_IF;

    L_Output.Confirmed_Closed := L_Valve.Confirmed_Closed;
    L_Output.Confirmed_Open := L_Valve.Confirmed_Open;
    L_Output.Confirmation_Unknown := L_Valve.Confirmation_Unknown;
    L_Output.Projection_Activated_Event := L_Output.Projection_Allowed;
    L_Output.Projection_Denied_Event := L_Output.Projection_Denied;

    GVL_Water_Output_Projection.G_Output_Projection_State[L_i] := L_Output;
    L_Any_Projected := L_Any_Projected OR L_Output.Projection_Allowed;
END_FOR;

GVL_Water_Output_Projection.G_Any_Output_Projected := L_Any_Projected;
GVL_Water_Output_Projection.G_Any_Projection_Denied := L_Any_Denied;
GVL_Water_Output_Projection.G_Global_Fallback_Projecting := L_Global_Fallback;
GVL_Water_Output_Projection.G_Runtime_Valid := TRUE;
GVL_Water_Output_Projection.G_Last_Update_MS := VI_System_Time_MS;

IF L_Global_Fallback THEN
    GVL_Water_Output_Projection.G_Status_Code := 2;
    GVL_Water_Output_Projection.G_Status_Text := 'Global fallback output projection active';
ELSIF L_Any_Projected THEN
    GVL_Water_Output_Projection.G_Status_Code := 1;
    GVL_Water_Output_Projection.G_Status_Text := 'Selective output projection active';
ELSE
    GVL_Water_Output_Projection.G_Status_Code := 0;
    GVL_Water_Output_Projection.G_Status_Text := 'No output projections active';
END_IF;
          
END_FUNCTION_BLOCK

FUNCTION_BLOCK FB_BlackBox_Recorder
  VAR_INPUT
    VI_Current_Data : ST_BlackBox_Record;
    VI_Freeze : BOOL;
  END_VAR
  VAR_OUTPUT
    VO_Frozen : BOOL;
    VO_Records_Count : INT;
  END_VAR
  VAR
    L_Write_Index : INT := 0;
    L_Initialized : BOOL := FALSE;
  END_VAR

            IF NOT L_Initialized THEN
    L_Write_Index := GVL_Retain.G_BlackBox_LastIndex;
    IF L_Write_Index < 0 OR L_Write_Index >= GVL_CONSTANTS.C_MAX_BLACKBOX_RECORDS THEN
        L_Write_Index := 0;
        GVL_Retain.G_BlackBox_LastIndex := 0;
    END_IF;
    L_Initialized := TRUE;
END_IF;

IF VI_Freeze THEN
    GVL_Retain.G_BlackBox_Frozen := TRUE;
END_IF;

VO_Frozen := GVL_Retain.G_BlackBox_Frozen;

IF NOT GVL_Retain.G_BlackBox_Frozen THEN
    GVL_Retain.G_BlackBox_Buffer[L_Write_Index] := VI_Current_Data;
    GVL_Retain.G_BlackBox_LastIndex := L_Write_Index;
    
    L_Write_Index := L_Write_Index + 1;
    IF L_Write_Index >= GVL_CONSTANTS.C_MAX_BLACKBOX_RECORDS THEN
        L_Write_Index := 0;
    END_IF;
END_IF;

VO_Records_Count := GVL_CONSTANTS.C_MAX_BLACKBOX_RECORDS; // Размер кольцевого буфера
// >>> BULK_SYNC_ANCHOR: FB_BlackBox_Recorder <<<
          
END_FUNCTION_BLOCK

FUNCTION_BLOCK FB_LogEvent
  VAR_INPUT
    VI_Event_Type : UINT;
    VI_Timestamp : UDINT;
    VI_Param1 : UDINT;
    VI_Param2 : UDINT;
  END_VAR

            GVL_EVENT.G_Event_Log[GVL_EVENT.G_Event_Head].Event_ID := GVL_EVENT.G_Event_ID_Counter;
GVL_EVENT.G_Event_Log[GVL_EVENT.G_Event_Head].Event_Type := VI_Event_Type;
GVL_EVENT.G_Event_Log[GVL_EVENT.G_Event_Head].Timestamp := VI_Timestamp;
GVL_EVENT.G_Event_Log[GVL_EVENT.G_Event_Head].Param1 := VI_Param1;
GVL_EVENT.G_Event_Log[GVL_EVENT.G_Event_Head].Param2 := VI_Param2;

GVL_EVENT.G_Event_ID_Counter := GVL_EVENT.G_Event_ID_Counter + 1;
GVL_EVENT.G_Event_Head := (GVL_EVENT.G_Event_Head + 1) MOD 64;
          
END_FUNCTION_BLOCK

FUNCTION_BLOCK FB_Heating_Schedule_Preheat
  VAR_INPUT
    VI_System_Time_MS : UDINT;
    VI_Time_Of_Day_MS : UDINT;
    VI_Day_Of_Week : INT;
    VI_Enable : BOOL;
  END_VAR
  VAR
    L_i : INT;
    L_e : INT;
    L_Event : ST_Heating_Schedule_Event;
    L_Time_To_Comfort_MS : UDINT;
    L_Adjustment : REAL;
    L_Max_Boost : REAL;
    L_Active : BOOL;
    L_Learn_Window_MS : UDINT := 300000;
    L_Learn_Cooldown_MS : UDINT := 900000;
    L_Cold_Confirm : ARRAY[1..GVL_CONSTANTS.C_MAX_ZONES, 1..3] OF INT;
    L_Hot_Confirm : ARRAY[1..GVL_CONSTANTS.C_MAX_ZONES, 1..3] OF INT;
    L_Last_Learn_MS : ARRAY[1..GVL_CONSTANTS.C_MAX_ZONES, 1..3] OF UDINT;
    L_Elapsed_MS : UDINT;
  END_VAR

            IF NOT VI_Enable THEN
    FOR L_i := 1 TO GVL_CONSTANTS.C_MAX_ZONES DO
        GVL_HEATING_POLICY.G_Zone_Schedule_Preheat_Active[L_i] := FALSE;
    END_FOR;
    RETURN;
END_IF;

FOR L_i := 1 TO GVL_CONSTANTS.C_MAX_ZONES DO
    L_Active := FALSE;
    L_Max_Boost := 0.0;

    FOR L_e := 1 TO 3 DO
        L_Event := GVL_HEATING_POLICY_CONFIG.G_Zone_Schedule[L_i, L_e];

        IF L_Event.Enabled THEN
            IF (L_Event.Weekday_Mask AND SHL(1, VI_Day_Of_Week - 1)) <> 0 THEN

                IF L_Event.Comfort_Time_MS >= VI_Time_Of_Day_MS THEN
                    L_Time_To_Comfort_MS := L_Event.Comfort_Time_MS - VI_Time_Of_Day_MS;
                ELSE
                    L_Time_To_Comfort_MS := (86400000 - VI_Time_Of_Day_MS) + L_Event.Comfort_Time_MS;
                END_IF;

                IF L_Event.Adaptive_Enabled THEN
                    IF GVL_HEATING_POLICY.G_Zone_Schedule_Learned_Offset_MS[L_i, L_e] > L_Event.Adaptive_Max_Offset_MS THEN
                        GVL_HEATING_POLICY.G_Zone_Schedule_Learned_Offset_MS[L_i, L_e] := L_Event.Adaptive_Max_Offset_MS;
                    END_IF;
                    L_Time_To_Comfort_MS := L_Time_To_Comfort_MS + GVL_HEATING_POLICY.G_Zone_Schedule_Learned_Offset_MS[L_i, L_e];
                END_IF;

                IF (GVL_HEATING_POLICY.G_Zone_Time_To_Heat_MS[L_i] >= L_Time_To_Comfort_MS)
                   AND (GVL_HEATING_POLICY.G_Zone_Time_To_Heat_MS[L_i] > 0) THEN

                    IF L_Event.Preheat_Boost > L_Max_Boost THEN
                        L_Max_Boost := L_Event.Preheat_Boost;
                    END_IF;

                    L_Active := TRUE;
                END_IF;

                IF L_Event.Adaptive_Enabled THEN
                    IF L_Time_To_Comfort_MS < L_Learn_Window_MS THEN

                        IF GVL_HEATING_POLICY.G_Zone_Thermal_Demand[L_i] > 1.0 THEN
                            L_Cold_Confirm[L_i, L_e] := L_Cold_Confirm[L_i, L_e] + 1;
                            L_Hot_Confirm[L_i, L_e] := 0;
                        ELSIF GVL_HEATING_POLICY.G_Zone_Thermal_Demand[L_i] < -0.5 THEN
                            L_Hot_Confirm[L_i, L_e] := L_Hot_Confirm[L_i, L_e] + 1;
                            L_Cold_Confirm[L_i, L_e] := 0;
                        ELSE
                            L_Cold_Confirm[L_i, L_e] := 0;
                            L_Hot_Confirm[L_i, L_e] := 0;
                        END_IF;

                        // UDINT wrap-safe elapsed time; unsigned subtraction is valid modulo 2^32.
                        L_Elapsed_MS := VI_System_Time_MS - L_Last_Learn_MS[L_i, L_e];

                        IF L_Elapsed_MS >= L_Learn_Cooldown_MS THEN

                            IF L_Cold_Confirm[L_i, L_e] >= 2 THEN
                                IF GVL_HEATING_POLICY.G_Zone_Schedule_Learned_Offset_MS[L_i, L_e] < L_Event.Adaptive_Max_Offset_MS THEN
                                    GVL_HEATING_POLICY.G_Zone_Schedule_Learned_Offset_MS[L_i, L_e] :=
                                        GVL_HEATING_POLICY.G_Zone_Schedule_Learned_Offset_MS[L_i, L_e] + L_Event.Adaptive_Step_MS;
                                    IF GVL_HEATING_POLICY.G_Zone_Schedule_Learned_Offset_MS[L_i, L_e] > L_Event.Adaptive_Max_Offset_MS THEN
                                        GVL_HEATING_POLICY.G_Zone_Schedule_Learned_Offset_MS[L_i, L_e] := L_Event.Adaptive_Max_Offset_MS;
                                    END_IF;
                                    L_Last_Learn_MS[L_i, L_e] := VI_System_Time_MS;
                                END_IF;
                                L_Cold_Confirm[L_i, L_e] := 0;
                            END_IF;

                            IF L_Hot_Confirm[L_i, L_e] >= 2 THEN
                                IF GVL_HEATING_POLICY.G_Zone_Schedule_Learned_Offset_MS[L_i, L_e] > L_Event.Adaptive_Step_MS THEN
                                    GVL_HEATING_POLICY.G_Zone_Schedule_Learned_Offset_MS[L_i, L_e] :=
                                        GVL_HEATING_POLICY.G_Zone_Schedule_Learned_Offset_MS[L_i, L_e] - L_Event.Adaptive_Step_MS;
                                ELSE
                                    GVL_HEATING_POLICY.G_Zone_Schedule_Learned_Offset_MS[L_i, L_e] := 0;
                                END_IF;
                                L_Last_Learn_MS[L_i, L_e] := VI_System_Time_MS;
                                L_Hot_Confirm[L_i, L_e] := 0;
                            END_IF;

                        END_IF;
                    ELSE
                        L_Cold_Confirm[L_i, L_e] := 0;
                        L_Hot_Confirm[L_i, L_e] := 0;
                    END_IF;
                END_IF;

            END_IF;
        END_IF;
    END_FOR;

    L_Adjustment := GVL_HEATING_POLICY.G_Zone_Target_Adjustment[L_i];

    IF L_Active AND (L_Adjustment < L_Max_Boost) THEN
        L_Adjustment := L_Max_Boost;
    END_IF;

    IF L_Adjustment > 1.0 THEN
        L_Adjustment := 1.0;
    ELSIF L_Adjustment < -1.0 THEN
        L_Adjustment := -1.0;
    END_IF;

    GVL_HEATING_POLICY.G_Zone_Target_Adjustment[L_i] := L_Adjustment;
    GVL_HEATING_POLICY.G_Zone_Schedule_Preheat_Active[L_i] := L_Active;
END_FOR;
          
END_FUNCTION_BLOCK

FUNCTION_BLOCK FB_Fault_Logger
  VAR_INPUT
    VI_Severity : E_System_Severity;
    VI_RootCause : E_System_Root_Cause;
    VI_Time_MS : UDINT;
  END_VAR
  VAR_OUTPUT
    VO_Last_Event_Text : STRING(200);
    VO_Event_Count : UINT;
    VO_Last_Index : UINT;
    VO_Event_Time_MS : ARRAY[1..16] OF UDINT;
    VO_Event_Severity : ARRAY[1..16] OF E_System_Severity;
    VO_Event_RootCause : ARRAY[1..16] OF E_System_Root_Cause;
    VO_Event_Text : ARRAY[1..16] OF STRING(200);
  END_VAR
  VAR
    L_Last_Severity : E_System_Severity;
    L_Last_RootCause : E_System_Root_Cause;
    L_Write_Index : UINT := 0;
    L_Event_Text : STRING(200);
  END_VAR

            L_Event_Text := '';

IF (VI_Severity <> L_Last_Severity) OR (VI_RootCause <> L_Last_RootCause) THEN
    CASE VI_RootCause OF
        E_System_Root_Cause.ROOT_FIRE:
            L_Event_Text := 'EVENT: FIRE DETECTED';
        E_System_Root_Cause.ROOT_GAS_LEAK:
            L_Event_Text := 'EVENT: GAS LEAK';
        E_System_Root_Cause.ROOT_CO_CRITICAL:
            L_Event_Text := 'EVENT: CO CRITICAL';
        E_System_Root_Cause.ROOT_CO_WARNING:
            L_Event_Text := 'EVENT: CO WARNING';
        E_System_Root_Cause.ROOT_WATER_LEAK:
            L_Event_Text := 'EVENT: WATER LEAK';
        E_System_Root_Cause.ROOT_SENSOR_FAULT:
            L_Event_Text := 'EVENT: SENSOR FAULT';
        E_System_Root_Cause.ROOT_IO_OFFLINE:
            L_Event_Text := 'EVENT: IO OFFLINE';
        E_System_Root_Cause.ROOT_COMM_FAULT:
            L_Event_Text := 'EVENT: COMM FAULT';
        E_System_Root_Cause.ROOT_WATCHDOG_FAULT:
            L_Event_Text := 'EVENT: WATCHDOG FAULT';
        E_System_Root_Cause.ROOT_SUBSYSTEM_FAULT:
            L_Event_Text := 'EVENT: SUBSYSTEM FAULT';
        ELSE
            L_Event_Text := 'EVENT: SYSTEM STATE CHANGE';
    END_CASE;

    L_Write_Index := L_Write_Index + 1;
    IF L_Write_Index > 16 THEN
        L_Write_Index := 1;
    END_IF;

    VO_Event_Time_MS[L_Write_Index] := VI_Time_MS;
    VO_Event_Severity[L_Write_Index] := VI_Severity;
    VO_Event_RootCause[L_Write_Index] := VI_RootCause;
    VO_Event_Text[L_Write_Index] := L_Event_Text;

    VO_Last_Index := L_Write_Index;
    VO_Last_Event_Text := L_Event_Text;

    IF VO_Event_Count < 16 THEN
        VO_Event_Count := VO_Event_Count + 1;
    END_IF;
END_IF;

L_Last_Severity := VI_Severity;
L_Last_RootCause := VI_RootCause;
// >>> BULK_SYNC_ANCHOR: FB_Fault_Logger <<<
          
END_FUNCTION_BLOCK

FUNCTION_BLOCK FB_Water_Hydraulic_Topology_Validator
  VAR_INPUT
    VI_Enable : BOOL;
    VI_System_Time_MS : UDINT;
  END_VAR
  VAR
    L_i : INT;
    L_Node : ST_Water_Hydraulic_Topology_Node;
    L_Group : ST_Water_Hydraulic_Isolation_Group;
    L_Validation : ST_Water_Topology_Validation_State;
    L_Empty_Node : ST_Water_Hydraulic_Topology_Node;
    L_Empty_Group : ST_Water_Hydraulic_Isolation_Group;
    L_Empty_Validation : ST_Water_Topology_Validation_State;
    L_Any_Invalid : BOOL;
    L_Any_Ambiguous : BOOL;
    L_Any_Fallback : BOOL;
  END_VAR

            IF NOT VI_Enable THEN
    GVL_Water_Topology_Validation.G_Runtime_Valid := FALSE;
    RETURN;
END_IF;

L_Any_Invalid := FALSE;
L_Any_Ambiguous := FALSE;
L_Any_Fallback := FALSE;

FOR L_i := 1 TO GVL_CONSTANTS.C_MAX_FLOOD_SENSORS DO

    L_Node := L_Empty_Node;
    L_Node.Runtime_Valid := TRUE;

    L_Node.Sensor_Id := TO_UINT(L_i);
    L_Node.Hydraulic_Zone_Id :=
        GVL_Water_Runtime_Projection.G_Leak_Runtime_State[L_i].Hydraulic_Zone_Id;

    L_Node.Valve_Group_Id :=
        GVL_Water_Runtime_Projection.G_Leak_Runtime_State[L_i].Valve_Group_Id;

    L_Node.Isolation_Group_Id :=
        L_Node.Valve_Group_Id;

    L_Node.Hydraulic_Segment_Id :=
        L_Node.Hydraulic_Zone_Id;

    L_Node.Fallback_Domain_Id := 1;

    // Validation.
    L_Node.Mapping_Valid :=
        L_Node.Valve_Group_Id <> 0;

    IF NOT L_Node.Mapping_Valid THEN
        L_Node.Global_Fallback_Required := TRUE;
        L_Node.Status_Code := 1;
        L_Node.Status_Text := 'Missing valve group';
    ELSE
        L_Node.Selective_Isolation_Allowed := TRUE;
        L_Node.Status_Code := 0;
        L_Node.Status_Text := 'Topology valid';
    END_IF;

    // Shared valve-group detection.
    IF L_Node.Valve_Group_Id = 3 THEN
        L_Node.Shared_Valve_Group := TRUE;
    END_IF;

    // Isolation group publication.
    L_Group := L_Empty_Group;
    L_Group.Runtime_Valid := TRUE;

    L_Group.Isolation_Group_Id :=
        L_Node.Isolation_Group_Id;

    L_Group.Valve_Group_Id :=
        L_Node.Valve_Group_Id;

    L_Group.Fallback_Domain_Id :=
        L_Node.Fallback_Domain_Id;

    L_Group.Shared_Sensor_Count :=
        SEL(L_Node.Shared_Valve_Group, 1, 2);

    L_Group.Isolation_Valid :=
        L_Node.Mapping_Valid;

    L_Group.Isolation_Ambiguous :=
        L_Node.Mapping_Ambiguous;

    L_Group.Selective_Isolation_Allowed :=
        L_Node.Selective_Isolation_Allowed;

    L_Group.Global_Fallback_Required :=
        L_Node.Global_Fallback_Required;

    // Validation publication.
    L_Validation := L_Empty_Validation;
    L_Validation.Runtime_Valid := TRUE;

    L_Validation.Runtime_System_Time_MS :=
        VI_System_Time_MS;

    L_Validation.Sensor_Id :=
        L_Node.Sensor_Id;

    L_Validation.Topology_Valid :=
        L_Node.Mapping_Valid;

    L_Validation.Topology_Ambiguous :=
        L_Node.Mapping_Ambiguous;

    L_Validation.Isolation_Path_Valid :=
        L_Group.Isolation_Valid;

    L_Validation.Shared_Valve_Group :=
        L_Node.Shared_Valve_Group;

    L_Validation.Missing_Valve_Group :=
        NOT L_Node.Mapping_Valid;

    L_Validation.Selective_Isolation_Allowed :=
        L_Node.Selective_Isolation_Allowed;

    L_Validation.Global_Fallback_Required :=
        L_Node.Global_Fallback_Required;

    IF L_Validation.Global_Fallback_Required THEN
        L_Validation.Status_Code := 1;
        L_Validation.Status_Text :=
            'Global fallback required';
    ELSE
        L_Validation.Status_Code := 0;
        L_Validation.Status_Text :=
            'Topology validation healthy';
    END_IF;

    GVL_Water_Hydraulic_Topology.G_Topology_Node[L_i] :=
        L_Node;

    GVL_Water_Hydraulic_Topology.G_Isolation_Group[L_i] :=
        L_Group;

    GVL_Water_Topology_Validation.G_Validation_State[L_i] :=
        L_Validation;

    L_Any_Invalid :=
        L_Any_Invalid
        OR NOT L_Validation.Topology_Valid;

    L_Any_Ambiguous :=
        L_Any_Ambiguous
        OR L_Validation.Topology_Ambiguous;

    L_Any_Fallback :=
        L_Any_Fallback
        OR L_Validation.Global_Fallback_Required;

END_FOR;

GVL_Water_Hydraulic_Topology.G_Any_Ambiguous :=
    L_Any_Ambiguous;

GVL_Water_Hydraulic_Topology.G_Any_Global_Fallback_Required :=
    L_Any_Fallback;

GVL_Water_Hydraulic_Topology.G_Runtime_Valid := TRUE;
GVL_Water_Hydraulic_Topology.G_Last_Update_MS := VI_System_Time_MS;

GVL_Water_Topology_Validation.G_Any_Invalid :=
    L_Any_Invalid;

GVL_Water_Topology_Validation.G_Any_Ambiguous :=
    L_Any_Ambiguous;

GVL_Water_Topology_Validation.G_Any_Global_Fallback_Required :=
    L_Any_Fallback;

GVL_Water_Topology_Validation.G_Runtime_Valid := TRUE;
GVL_Water_Topology_Validation.G_Last_Update_MS := VI_System_Time_MS;
          
END_FUNCTION_BLOCK

FUNCTION_BLOCK FB_Watchdog
  VAR_INPUT
    VI_System_Time_MS : UDINT;
    VI_Timeout_MS : UDINT := 2000;
  END_VAR
  VAR_OUTPUT
    VO_Alive : BOOL;
    VO_Watchdog_Fault : BOOL;
    VO_Cycle_DT_MS : UDINT;
  END_VAR
  VAR
    L_Initialized : BOOL := FALSE;
    L_Last_Call_MS : UDINT := 0;
    L_DT_MS : UDINT := 0;
  END_VAR

            IF NOT L_Initialized THEN
    L_Initialized := TRUE;
    L_Last_Call_MS := VI_System_Time_MS;
    VO_Cycle_DT_MS := 0;
    VO_Watchdog_Fault := FALSE;
    VO_Alive := TRUE;
    RETURN;
END_IF;

// Measure real time gap between successive calls
L_DT_MS := (SEL(VI_System_Time_MS >= L_Last_Call_MS, VI_System_Time_MS - L_Last_Call_MS, (4294967295 - L_Last_Call_MS) + VI_System_Time_MS + 1));
VO_Cycle_DT_MS := L_DT_MS;

// Fault if the task/cycle resumed after an abnormal pause
VO_Watchdog_Fault := (L_DT_MS > VI_Timeout_MS);
VO_Alive := NOT VO_Watchdog_Fault;

// Store current timestamp for next cycle
L_Last_Call_MS := VI_System_Time_MS;
// >>> BULK_SYNC_ANCHOR: FB_Watchdog <<<
          
END_FUNCTION_BLOCK

FUNCTION_BLOCK FB_Socket_Manager
  VAR_INPUT
    VI_System_Time_MS : UDINT;
    VI_IsActivePLC : BOOL;
    VI_Scenario : E_SCENARIO_TYPE;
    VI_Fire_Alarm : BOOL;
    VI_Flood_Alarm : BOOL;
    VI_Security_Armed : BOOL;
  END_VAR
  VAR_OUTPUT
    VO_Socket_States : ARRAY[1..GVL_CONSTANTS.C_MAX_SOCKETS] OF BOOL;
    VO_Internal_States : ARRAY[1..GVL_CONSTANTS.C_MAX_SOCKETS] OF BOOL;
  END_VAR
  VAR_IN_OUT
    VI_Manual_Override : ARRAY[1..GVL_CONSTANTS.C_MAX_SOCKETS] OF BOOL;
    VI_Physical_Switches : ARRAY[1..GVL_CONSTANTS.C_MAX_SOCKETS] OF BOOL;
    VI_Rule_Actions : ARRAY[1..GVL_CONSTANTS.C_MAX_RULES] OF ST_Rule_Action;
    VI_IO_Modules_Online : ARRAY[1..GVL_CONSTANTS.C_MAX_MODULES] OF BOOL;
  END_VAR
  VAR
    L_i : INT;
    L_j : INT;
    L_Rule_State : BOOL;
    L_Rule_Active : BOOL;
    L_Internal_State : ARRAY[1..GVL_CONSTANTS.C_MAX_SOCKETS] OF BOOL;
    L_Manual_Trig : ARRAY[1..GVL_CONSTANTS.C_MAX_SOCKETS] OF R_TRIG;
  END_VAR

            // Менеджер управления розетками.
// Обеспечивает работу по сценариям, правилам и аварийное отключение (без локальных выключателей розеток).


IF NOT VI_IsActivePLC THEN RETURN; END_IF;


// Проверка связи с модулями ввода-вывода
FOR L_i := 1 TO GVL_CONSTANTS.C_MAX_MODULES DO
    IF NOT VI_IO_Modules_Online[L_i] THEN
        // Переход в безопасное состояние при потере связи (отключение всех розеток)
        FOR L_j := 1 TO GVL_CONSTANTS.C_MAX_SOCKETS DO
            VO_Socket_States[L_j] := FALSE;
        END_FOR;
        RETURN;
    END_IF;
END_FOR;

FOR L_i := 1 TO GVL_CONSTANTS.C_MAX_SOCKETS DO
    L_Rule_Active := FALSE;
    L_Rule_State := FALSE;
    
    L_Manual_Trig[L_i](CLK := VI_Manual_Override[L_i]);
    
    // Ручное переключение
    IF L_Manual_Trig[L_i].Q THEN
        L_Internal_State[L_i] := NOT L_Internal_State[L_i];
    END_IF;

    // Проверка правил для текущей розетки
    FOR L_j := 1 TO GVL_CONSTANTS.C_MAX_RULES DO
        IF VI_Rule_Actions[L_j].Active AND VI_Rule_Actions[L_j].Target_ID = L_i THEN
            IF VI_Rule_Actions[L_j].Action_Type = E_Rule_Action_Type.ACTION_SET_SOCKET THEN
                L_Rule_Active := TRUE;
                L_Rule_State := (VI_Rule_Actions[L_j].Value > 0.5);
                L_Internal_State[L_i] := L_Rule_State; // Синхронизация внутреннего состояния
            ELSIF VI_Rule_Actions[L_j].Action_Type = E_Rule_Action_Type.ACTION_TOGGLE_SOCKET AND VI_Rule_Actions[L_j].Triggered THEN
                L_Internal_State[L_i] := NOT L_Internal_State[L_i]; // Toggle
            END_IF;
        END_IF;
    END_FOR;

    // Аварийное отключение
    IF VI_Fire_Alarm OR VI_Flood_Alarm THEN
        // Розетки 1-4 неотключаемые (холодильник, сервер и т.д.)
        IF L_i > 4 THEN
            VO_Socket_States[L_i] := FALSE;
        ELSE
            // Критические розетки сохраняют свое текущее внутреннее состояние, а не форсируются в TRUE
            VO_Socket_States[L_i] := L_Internal_State[L_i];
        END_IF;
    ELSIF VI_Scenario = E_SCENARIO_TYPE.SCENARIO_AWAY OR VI_Security_Armed THEN
        // Master Off
        IF L_i > 4 THEN
            VO_Socket_States[L_i] := FALSE;
        ELSE
            // Неотключаемые розетки могут управляться вручную
            VO_Socket_States[L_i] := L_Internal_State[L_i];
        END_IF;
    ELSE
        // Нормальный режим: состояние определяется внутренним состоянием (ручным или правилом)
        IF L_Rule_Active THEN
            VO_Socket_States[L_i] := L_Rule_State;
        ELSE
            VO_Socket_States[L_i] := L_Internal_State[L_i];
        END_IF;
    END_IF;
END_FOR;

VO_Internal_States := L_Internal_State;

// >>> BULK_SYNC_ANCHOR: FB_Socket_Manager <<<
          
END_FUNCTION_BLOCK

FUNCTION_BLOCK FB_System_Health
  VAR_INPUT
    VI_Smoke_Detected : BOOL;
    VI_Gas_Detected : BOOL;
    VI_CO_Warning_Level : BOOL;
    VI_CO_Alarm_Level : BOOL;
    VI_Leak_Detected : BOOL;
    VI_Sensor_Fault : BOOL := FALSE;
    VI_IO_Offline : BOOL := FALSE;
    VI_Comm_Fault : BOOL := FALSE;
    VI_Watchdog_Fault : BOOL := FALSE;
    VI_Subsystem_Fault : BOOL := FALSE;
  END_VAR
  VAR_OUTPUT
    VO_System_Severity : E_System_Severity;
    VO_Root_Cause : E_System_Root_Cause;
    VO_Sensor_Fault : BOOL;
    VO_IO_Fault : BOOL;
    VO_Comm_Fault : BOOL;
    VO_Subsystem_Degraded : BOOL;
    VO_First_Fault_Active : BOOL;
    VO_First_Fault_Type : INT;
    VO_First_Fault_Source : INT;
    VO_IO_Fault_Count : UDINT;
    VO_Comm_Fault_Count : UDINT;
    VO_Sensor_Fault_Count : UDINT;
    VO_Subsystem_Fault_Count : UDINT;
    VO_Watchdog_Fault_Count : UDINT;
  END_VAR
  VAR
    L_IO_Fault_Assert_Count : UINT;
    L_IO_Fault_Clear_Count : UINT;
    L_IO_Fault_Stable : BOOL;
    L_Comm_Fault_Assert_Count : UINT;
    L_Comm_Fault_Clear_Count : UINT;
    L_Comm_Fault_Stable : BOOL;
    L_Sensor_Fault_Assert_Count : UINT;
    L_Sensor_Fault_Clear_Count : UINT;
    L_Sensor_Fault_Stable : BOOL;
    L_Subsystem_Assert_Count : UINT;
    L_Subsystem_Clear_Count : UINT;
    L_Subsystem_Fault_Stable : BOOL;
    L_IO_Fault_Prev : BOOL;
    L_Comm_Fault_Prev : BOOL;
    L_Sensor_Fault_Prev : BOOL;
    L_Subsystem_Fault_Prev : BOOL;
    L_Watchdog_Fault_Prev : BOOL;
  END_VAR
  VAR CONSTANT
    C_HEALTH_DEBOUNCE_CYCLES : UINT := 3;
  END_VAR

            // Debounce non-critical diagnostics: require 3 stable cycles to assert/clear
IF VI_IO_Offline THEN
    L_IO_Fault_Clear_Count := 0;
    IF L_IO_Fault_Assert_Count < C_HEALTH_DEBOUNCE_CYCLES THEN
        L_IO_Fault_Assert_Count := L_IO_Fault_Assert_Count + 1;
    END_IF;
    IF L_IO_Fault_Assert_Count >= C_HEALTH_DEBOUNCE_CYCLES THEN
        L_IO_Fault_Stable := TRUE;
    END_IF;
ELSE
    L_IO_Fault_Assert_Count := 0;
    IF L_IO_Fault_Clear_Count < C_HEALTH_DEBOUNCE_CYCLES THEN
        L_IO_Fault_Clear_Count := L_IO_Fault_Clear_Count + 1;
    END_IF;
    IF L_IO_Fault_Clear_Count >= C_HEALTH_DEBOUNCE_CYCLES THEN
        L_IO_Fault_Stable := FALSE;
    END_IF;
END_IF;

IF VI_Comm_Fault THEN
    L_Comm_Fault_Clear_Count := 0;
    IF L_Comm_Fault_Assert_Count < C_HEALTH_DEBOUNCE_CYCLES THEN
        L_Comm_Fault_Assert_Count := L_Comm_Fault_Assert_Count + 1;
    END_IF;
    IF L_Comm_Fault_Assert_Count >= C_HEALTH_DEBOUNCE_CYCLES THEN
        L_Comm_Fault_Stable := TRUE;
    END_IF;
ELSE
    L_Comm_Fault_Assert_Count := 0;
    IF L_Comm_Fault_Clear_Count < C_HEALTH_DEBOUNCE_CYCLES THEN
        L_Comm_Fault_Clear_Count := L_Comm_Fault_Clear_Count + 1;
    END_IF;
    IF L_Comm_Fault_Clear_Count >= C_HEALTH_DEBOUNCE_CYCLES THEN
        L_Comm_Fault_Stable := FALSE;
    END_IF;
END_IF;

